LIN {X 2.525,Y 79.377,Z 54.000,A 180.000,B 0.000,C 180.000} C_DIS
LIN {X 2.581,Y 80.986,Z 54.000,A 180.000,B 0.000,C 180.000} C_DIS
LIN {X 2.591,Y 81.165,Z 54.000,A 180.000,B 0.000,C 180.000} C_DIS
LIN {X 2.675,Y 82.595,Z 54.000,A 180.000,B 0.000,C 180.000} C_DIS
LIN {X 2.685,Y 82.761,Z 54.000,A 180.000,B 0.000,C 180.000} C_DIS
LIN {X 2.686,Y 82.774,Z 54.000,A 180.000,B 0.000,C 180.000} C_DIS
LIN {X 2.700,Y 82.952,Z 54.000,A 180.000,B 0.000,C 180.000} C_DIS
LIN {X 2.818,Y 84.383,Z 54.000,A 180.000,B 0.000,C 180.000} C_DIS
LIN {X 2.833,Y 84.561,Z 54.000,A 180.000,B 0.000,C 180.000} C_DIS
LIN {X 3.004,Y 86.170,Z 54.000,A 180.000,B 0.000,C 180.000} C_DIS
LIN {X 3.025,Y 86.349,Z 54.000,A 180.000,B 0.000,C 180.000} C_DIS
LIN {X 3.233,Y 87.958,Z 54.000,A 180.000,B 0.000,C 180.000} C_DIS
LIN {X 3.259,Y 88.137,Z 54.000,A 180.000,B 0.000,C 180.000} C_DIS
LIN {X 3.479,Y 89.567,Z 54.000,A 180.000,B 0.000,C 180.000} C_DIS
LIN {X 3.506,Y 89.746,Z 54.000,A 180.000,B 0.000,C 180.000} C_DIS
LIN {X 3.538,Y 89.925,Z 54.000,A 180.000,B 0.000,C 180.000} C_DIS
LIN {X 3.792,Y 91.355,Z 54.000,A 180.000,B 0.000,C 180.000} C_DIS
LIN {X 3.825,Y 91.533,Z 54.000,A 180.000,B 0.000,C 180.000} C_DIS
LIN {X 4.150,Y 93.142,Z 54.000,A 180.000,B 0.000,C 180.000} C_DIS
LIN {X 4.189,Y 93.321,Z 54.000,A 180.000,B 0.000,C 180.000} C_DIS
LIN {X 4.513,Y 94.751,Z 54.000,A 180.000,B 0.000,C 180.000} C_DIS
LIN {X 4.554,Y 94.930,Z 54.000,A 180.000,B 0.000,C 180.000} C_DIS
LIN {X 4.598,Y 95.109,Z 54.000,A 180.000,B 0.000,C 180.000} C_DIS
LIN {X 4.958,Y 96.539,Z 54.000,A 180.000,B 0.000,C 180.000} C_DIS
LIN {X 5.005,Y 96.718,Z 54.000,A 180.000,B 0.000,C 180.000} C_DIS
LIN {X 5.400,Y 98.148,Z 54.000,A 180.000,B 0.000,C 180.000} C_DIS
LIN {X 5.450,Y 98.327,Z 54.000,A 180.000,B 0.000,C 180.000} C_DIS
LIN {X 5.503,Y 98.505,Z 54.000,A 180.000,B 0.000,C 180.000} C_DIS
LIN {X 5.935,Y 99.936,Z 54.000,A 180.000,B 0.000,C 180.000} C_DIS
LIN {X 5.992,Y 100.114,Z 54.000,A 180.000,B 0.000,C 180.000} C_DIS
LIN {X 6.460,Y 101.545,Z 54.000,A 180.000,B 0.000,C 180.000} C_DIS
LIN {X 6.520,Y 101.723,Z 54.000,A 180.000,B 0.000,C 180.000} C_DIS
LIN {X 7.026,Y 103.153,Z 54.000,A 180.000,B 0.000,C 180.000} C_DIS
LIN {X 7.089,Y 103.332,Z 54.000,A 180.000,B 0.000,C 180.000} C_DIS
LIN {X 7.154,Y 103.504,Z 54.000,A 180.000,B 0.000,C 180.000} C_DIS
LIN {X 7.701,Y 104.941,Z 54.000,A 180.000,B 0.000,C 180.000} C_DIS
LIN {X 7.773,Y 105.120,Z 54.000,A 180.000,B 0.000,C 180.000} C_DIS
LIN {X 8.355,Y 106.550,Z 54.000,A 180.000,B 0.000,C 180.000} C_DIS
LIN {X 8.405,Y 106.669,Z 54.000,A 180.000,B 0.000,C 180.000} C_DIS
LIN {X 9.053,Y 108.159,Z 54.000,A 180.000,B 0.000,C 180.000} C_DIS
LIN {X 9.120,Y 108.308,Z 54.000,A 180.000,B 0.000,C 180.000} C_DIS
LIN {X 9.797,Y 109.768,Z 54.000,A 180.000,B 0.000,C 180.000} C_DIS
LIN {X 9.836,Y 109.849,Z 54.000,A 180.000,B 0.000,C 180.000} C_DIS
LIN {X 10.551,Y 111.303,Z 54.000,A 180.000,B 0.000,C 180.000} C_DIS
LIN {X 10.587,Y 111.377,Z 54.000,A 180.000,B 0.000,C 180.000} C_DIS
LIN {X 10.680,Y 111.556,Z 54.000,A 180.000,B 0.000,C 180.000} C_DIS
LIN {X 11.332,Y 112.807,Z 54.000,A 180.000,B 0.000,C 180.000} C_DIS
LIN {X 11.426,Y 112.986,Z 54.000,A 180.000,B 0.000,C 180.000} C_DIS
LIN {X 12.215,Y 114.416,Z 54.000,A 180.000,B 0.000,C 180.000} C_DIS
LIN {X 12.317,Y 114.595,Z 54.000,A 180.000,B 0.000,C 180.000} C_DIS
LIN {X 13.053,Y 115.859,Z 54.000,A 180.000,B 0.000,C 180.000} C_DIS
LIN {X 13.151,Y 116.025,Z 54.000,A 180.000,B 0.000,C 180.000} C_DIS
LIN {X 13.232,Y 116.158,Z 54.000,A 180.000,B 0.000,C 180.000} C_DIS
LIN {X 14.029,Y 117.455,Z 54.000,A 180.000,B 0.000,C 180.000} C_DIS
LIN {X 14.126,Y 117.607,Z 54.000,A 180.000,B 0.000,C 180.000} C_DIS
LIN {X 14.953,Y 118.885,Z 54.000,A 180.000,B 0.000,C 180.000} C_DIS
LIN {X 15.020,Y 118.988,Z 54.000,A 180.000,B 0.000,C 180.000} C_DIS
LIN {X 15.072,Y 119.064,Z 54.000,A 180.000,B 0.000,C 180.000} C_DIS
LIN {X 15.924,Y 120.315,Z 54.000,A 180.000,B 0.000,C 180.000} C_DIS
LIN {X 16.047,Y 120.494,Z 54.000,A 180.000,B 0.000,C 180.000} C_DIS
LIN {X 16.986,Y 121.806,Z 54.000,A 180.000,B 0.000,C 180.000} C_DIS
LIN {X 17.073,Y 121.924,Z 54.000,A 180.000,B 0.000,C 180.000} C_DIS
LIN {X 18.059,Y 123.235,Z 54.000,A 180.000,B 0.000,C 180.000} C_DIS
LIN {X 18.152,Y 123.354,Z 54.000,A 180.000,B 0.000,C 180.000} C_DIS
LIN {X 19.139,Y 124.606,Z 54.000,A 180.000,B 0.000,C 180.000} C_DIS
LIN {X 19.286,Y 124.785,Z 54.000,A 180.000,B 0.000,C 180.000} C_DIS
LIN {X 20.204,Y 125.894,Z 54.000,A 180.000,B 0.000,C 180.000} C_DIS
LIN {X 20.323,Y 126.036,Z 54.000,A 180.000,B 0.000,C 180.000} C_DIS
LIN {X 21.410,Y 127.287,Z 54.000,A 180.000,B 0.000,C 180.000} C_DIS
LIN {X 21.456,Y 127.340,Z 54.000,A 180.000,B 0.000,C 180.000} C_DIS
LIN {X 21.570,Y 127.466,Z 54.000,A 180.000,B 0.000,C 180.000} C_DIS
LIN {X 22.547,Y 128.539,Z 54.000,A 180.000,B 0.000,C 180.000} C_DIS
LIN {X 22.707,Y 128.711,Z 54.000,A 180.000,B 0.000,C 180.000} C_DIS
LIN {X 23.780,Y 129.835,Z 54.000,A 180.000,B 0.000,C 180.000} C_DIS
LIN {X 23.910,Y 129.969,Z 54.000,A 180.000,B 0.000,C 180.000} C_DIS
LIN {X 25.031,Y 131.090,Z 54.000,A 180.000,B 0.000,C 180.000} C_DIS
LIN {X 25.165,Y 131.220,Z 54.000,A 180.000,B 0.000,C 180.000} C_DIS
LIN {X 26.289,Y 132.293,Z 54.000,A 180.000,B 0.000,C 180.000} C_DIS
LIN {X 26.461,Y 132.453,Z 54.000,A 180.000,B 0.000,C 180.000} C_DIS
LIN {X 27.534,Y 133.430,Z 54.000,A 180.000,B 0.000,C 180.000} C_DIS
LIN {X 27.660,Y 133.544,Z 54.000,A 180.000,B 0.000,C 180.000} C_DIS
LIN {X 27.713,Y 133.590,Z 54.000,A 180.000,B 0.000,C 180.000} C_DIS
LIN {X 28.964,Y 134.677,Z 54.000,A 180.000,B 0.000,C 180.000} C_DIS
LIN {X 29.106,Y 134.796,Z 54.000,A 180.000,B 0.000,C 180.000} C_DIS
LIN {X 30.215,Y 135.714,Z 54.000,A 180.000,B 0.000,C 180.000} C_DIS
LIN {X 30.394,Y 135.861,Z 54.000,A 180.000,B 0.000,C 180.000} C_DIS
LIN {X 31.646,Y 136.848,Z 54.000,A 180.000,B 0.000,C 180.000} C_DIS
LIN {X 31.765,Y 136.941,Z 54.000,A 180.000,B 0.000,C 180.000} C_DIS
LIN {X 33.076,Y 137.927,Z 54.000,A 180.000,B 0.000,C 180.000} C_DIS
LIN {X 33.194,Y 138.014,Z 54.000,A 180.000,B 0.000,C 180.000} C_DIS
LIN {X 34.506,Y 138.953,Z 54.000,A 180.000,B 0.000,C 180.000} C_DIS
LIN {X 34.685,Y 139.076,Z 54.000,A 180.000,B 0.000,C 180.000} C_DIS
LIN {X 35.936,Y 139.928,Z 54.000,A 180.000,B 0.000,C 180.000} C_DIS
LIN {X 36.012,Y 139.980,Z 54.000,A 180.000,B 0.000,C 180.000} C_DIS
LIN {X 36.115,Y 140.047,Z 54.000,A 180.000,B 0.000,C 180.000} C_DIS
LIN {X 37.393,Y 140.874,Z 54.000,A 180.000,B 0.000,C 180.000} C_DIS
LIN {X 37.545,Y 140.971,Z 54.000,A 180.000,B 0.000,C 180.000} C_DIS
LIN {X 38.842,Y 141.768,Z 54.000,A 180.000,B 0.000,C 180.000} C_DIS
LIN {X 38.975,Y 141.849,Z 54.000,A 180.000,B 0.000,C 180.000} C_DIS
LIN {X 39.141,Y 141.947,Z 54.000,A 180.000,B 0.000,C 180.000} C_DIS
LIN {X 40.405,Y 142.683,Z 54.000,A 180.000,B 0.000,C 180.000} C_DIS
LIN {X 40.584,Y 142.785,Z 54.000,A 180.000,B 0.000,C 180.000} C_DIS
LIN {X 42.014,Y 143.574,Z 54.000,A 180.000,B 0.000,C 180.000} C_DIS
LIN {X 42.193,Y 143.668,Z 54.000,A 180.000,B 0.000,C 180.000} C_DIS
LIN {X 43.444,Y 144.320,Z 54.000,A 180.000,B 0.000,C 180.000} C_DIS
LIN {X 43.623,Y 144.413,Z 54.000,A 180.000,B 0.000,C 180.000} C_DIS
LIN {X 43.697,Y 144.449,Z 54.000,A 180.000,B 0.000,C 180.000} C_DIS
LIN {X 45.151,Y 145.164,Z 54.000,A 180.000,B 0.000,C 180.000} C_DIS
LIN {X 45.232,Y 145.203,Z 54.000,A 180.000,B 0.000,C 180.000} C_DIS
LIN {X 46.692,Y 145.880,Z 54.000,A 180.000,B 0.000,C 180.000} C_DIS
LIN {X 46.841,Y 145.947,Z 54.000,A 180.000,B 0.000,C 180.000} C_DIS
LIN {X 48.331,Y 146.595,Z 54.000,A 180.000,B 0.000,C 180.000} C_DIS
LIN {X 48.450,Y 146.645,Z 54.000,A 180.000,B 0.000,C 180.000} C_DIS
LIN {X 49.880,Y 147.227,Z 54.000,A 180.000,B 0.000,C 180.000} C_DIS
LIN {X 50.059,Y 147.299,Z 54.000,A 180.000,B 0.000,C 180.000} C_DIS
LIN {X 51.496,Y 147.846,Z 54.000,A 180.000,B 0.000,C 180.000} C_DIS
LIN {X 51.668,Y 147.911,Z 54.000,A 180.000,B 0.000,C 180.000} C_DIS
LIN {X 51.847,Y 147.974,Z 54.000,A 180.000,B 0.000,C 180.000} C_DIS
LIN {X 53.277,Y 148.480,Z 54.000,A 180.000,B 0.000,C 180.000} C_DIS
LIN {X 53.455,Y 148.540,Z 54.000,A 180.000,B 0.000,C 180.000} C_DIS
LIN {X 54.290,Y 148.813,Z 54.000,A 180.000,B 0.000,C 180.000} C_DIS
LIN {X 54.886,Y 149.008,Z 54.000,A 180.000,B 0.000,C 180.000} C_DIS
LIN {X 55.064,Y 149.065,Z 54.000,A 180.000,B 0.000,C 180.000} C_DIS
LIN {X 56.495,Y 149.497,Z 54.000,A 180.000,B 0.000,C 180.000} C_DIS
LIN {X 56.673,Y 149.550,Z 54.000,A 180.000,B 0.000,C 180.000} C_DIS
LIN {X 56.852,Y 149.600,Z 54.000,A 180.000,B 0.000,C 180.000} C_DIS
LIN {X 58.282,Y 149.995,Z 54.000,A 180.000,B 0.000,C 180.000} C_DIS
LIN {X 58.461,Y 150.042,Z 54.000,A 180.000,B 0.000,C 180.000} C_DIS
LIN {X 59.891,Y 150.402,Z 54.000,A 180.000,B 0.000,C 180.000} C_DIS
LIN {X 60.070,Y 150.447,Z 54.000,A 180.000,B 0.000,C 180.000} C_DIS
LIN {X 60.249,Y 150.487,Z 54.000,A 180.000,B 0.000,C 180.000} C_DIS
LIN {X 61.679,Y 150.811,Z 54.000,A 180.000,B 0.000,C 180.000} C_DIS
LIN {X 61.858,Y 150.850,Z 54.000,A 180.000,B 0.000,C 180.000} C_DIS
LIN {X 63.467,Y 151.175,Z 54.000,A 180.000,B 0.000,C 180.000} C_DIS
LIN {X 63.645,Y 151.208,Z 54.000,A 180.000,B 0.000,C 180.000} C_DIS
LIN {X 65.075,Y 151.462,Z 54.000,A 180.000,B 0.000,C 180.000} C_DIS
LIN {X 65.254,Y 151.494,Z 54.000,A 180.000,B 0.000,C 180.000} C_DIS
LIN {X 65.433,Y 151.521,Z 54.000,A 180.000,B 0.000,C 180.000} C_DIS
LIN {X 66.863,Y 151.741,Z 54.000,A 180.000,B 0.000,C 180.000} C_DIS
LIN {X 67.042,Y 151.767,Z 54.000,A 180.000,B 0.000,C 180.000} C_DIS
LIN {X 68.651,Y 151.975,Z 54.000,A 180.000,B 0.000,C 180.000} C_DIS
LIN {X 68.830,Y 151.996,Z 54.000,A 180.000,B 0.000,C 180.000} C_DIS
LIN {X 70.439,Y 152.167,Z 54.000,A 180.000,B 0.000,C 180.000} C_DIS
LIN {X 70.617,Y 152.182,Z 54.000,A 180.000,B 0.000,C 180.000} C_DIS
LIN {X 72.048,Y 152.300,Z 54.000,A 180.000,B 0.000,C 180.000} C_DIS
LIN {X 72.226,Y 152.314,Z 54.000,A 180.000,B 0.000,C 180.000} C_DIS
LIN {X 72.239,Y 152.315,Z 54.000,A 180.000,B 0.000,C 180.000} C_DIS
LIN {X 72.405,Y 152.325,Z 54.000,A 180.000,B 0.000,C 180.000} C_DIS
LIN {X 73.835,Y 152.409,Z 54.000,A 180.000,B 0.000,C 180.000} C_DIS
LIN {X 74.014,Y 152.419,Z 54.000,A 180.000,B 0.000,C 180.000} C_DIS
LIN {X 75.623,Y 152.475,Z 54.000,A 180.000,B 0.000,C 180.000} C_DIS
LIN {X 75.802,Y 152.480,Z 54.000,A 180.000,B 0.000,C 180.000} C_DIS
LIN {X 77.411,Y 152.499,Z 54.000,A 180.000,B 0.000,C 180.000} C_DIS
LIN {X 77.589,Y 152.499,Z 54.000,A 180.000,B 0.000,C 180.000} C_DIS
LIN {X 79.198,Y 152.480,Z 54.000,A 180.000,B 0.000,C 180.000} C_DIS
LIN {X 79.377,Y 152.475,Z 54.000,A 180.000,B 0.000,C 180.000} C_DIS
LIN {X 80.986,Y 152.419,Z 54.000,A 180.000,B 0.000,C 180.000} C_DIS
LIN {X 81.165,Y 152.409,Z 54.000,A 180.000,B 0.000,C 180.000} C_DIS
LIN {X 82.595,Y 152.325,Z 54.000,A 180.000,B 0.000,C 180.000} C_DIS
LIN {X 82.761,Y 152.315,Z 54.000,A 180.000,B 0.000,C 180.000} C_DIS
LIN {X 82.774,Y 152.314,Z 54.000,A 180.000,B 0.000,C 180.000} C_DIS
LIN {X 82.952,Y 152.300,Z 54.000,A 180.000,B 0.000,C 180.000} C_DIS
LIN {X 84.383,Y 152.182,Z 54.000,A 180.000,B 0.000,C 180.000} C_DIS
LIN {X 84.561,Y 152.167,Z 54.000,A 180.000,B 0.000,C 180.000} C_DIS
LIN {X 86.170,Y 151.996,Z 54.000,A 180.000,B 0.000,C 180.000} C_DIS
LIN {X 86.349,Y 151.975,Z 54.000,A 180.000,B 0.000,C 180.000} C_DIS
LIN {X 87.958,Y 151.767,Z 54.000,A 180.000,B 0.000,C 180.000} C_DIS
LIN {X 88.137,Y 151.741,Z 54.000,A 180.000,B 0.000,C 180.000} C_DIS
LIN {X 89.567,Y 151.521,Z 54.000,A 180.000,B 0.000,C 180.000} C_DIS
LIN {X 89.746,Y 151.494,Z 54.000,A 180.000,B 0.000,C 180.000} C_DIS
LIN {X 89.925,Y 151.462,Z 54.000,A 180.000,B 0.000,C 180.000} C_DIS
LIN {X 91.355,Y 151.208,Z 54.000,A 180.000,B 0.000,C 180.000} C_DIS
LIN {X 91.533,Y 151.175,Z 54.000,A 180.000,B 0.000,C 180.000} C_DIS
LIN {X 93.142,Y 150.850,Z 54.000,A 180.000,B 0.000,C 180.000} C_DIS
LIN {X 93.321,Y 150.811,Z 54.000,A 180.000,B 0.000,C 180.000} C_DIS
LIN {X 94.751,Y 150.487,Z 54.000,A 180.000,B 0.000,C 180.000} C_DIS
LIN {X 94.930,Y 150.447,Z 54.000,A 180.000,B 0.000,C 180.000} C_DIS
LIN {X 95.109,Y 150.402,Z 54.000,A 180.000,B 0.000,C 180.000} C_DIS
LIN {X 96.539,Y 150.042,Z 54.000,A 180.000,B 0.000,C 180.000} C_DIS
LIN {X 96.718,Y 149.995,Z 54.000,A 180.000,B 0.000,C 180.000} C_DIS
LIN {X 98.148,Y 149.600,Z 54.000,A 180.000,B 0.000,C 180.000} C_DIS
LIN {X 98.327,Y 149.550,Z 54.000,A 180.000,B 0.000,C 180.000} C_DIS
LIN {X 98.505,Y 149.497,Z 54.000,A 180.000,B 0.000,C 180.000} C_DIS
LIN {X 99.936,Y 149.065,Z 54.000,A 180.000,B 0.000,C 180.000} C_DIS
LIN {X 100.114,Y 149.008,Z 54.000,A 180.000,B 0.000,C 180.000} C_DIS
LIN {X 101.545,Y 148.540,Z 54.000,A 180.000,B 0.000,C 180.000} C_DIS
LIN {X 101.723,Y 148.480,Z 54.000,A 180.000,B 0.000,C 180.000} C_DIS
LIN {X 103.153,Y 147.974,Z 54.000,A 180.000,B 0.000,C 180.000} C_DIS
LIN {X 103.332,Y 147.911,Z 54.000,A 180.000,B 0.000,C 180.000} C_DIS
LIN {X 103.504,Y 147.846,Z 54.000,A 180.000,B 0.000,C 180.000} C_DIS
LIN {X 104.941,Y 147.299,Z 54.000,A 180.000,B 0.000,C 180.000} C_DIS
LIN {X 105.120,Y 147.227,Z 54.000,A 180.000,B 0.000,C 180.000} C_DIS
LIN {X 106.550,Y 146.645,Z 54.000,A 180.000,B 0.000,C 180.000} C_DIS
LIN {X 106.669,Y 146.595,Z 54.000,A 180.000,B 0.000,C 180.000} C_DIS
LIN {X 108.159,Y 145.947,Z 54.000,A 180.000,B 0.000,C 180.000} C_DIS
LIN {X 108.308,Y 145.880,Z 54.000,A 180.000,B 0.000,C 180.000} C_DIS
LIN {X 109.768,Y 145.203,Z 54.000,A 180.000,B 0.000,C 180.000} C_DIS
LIN {X 109.849,Y 145.164,Z 54.000,A 180.000,B 0.000,C 180.000} C_DIS
LIN {X 111.303,Y 144.449,Z 54.000,A 180.000,B 0.000,C 180.000} C_DIS
LIN {X 111.377,Y 144.413,Z 54.000,A 180.000,B 0.000,C 180.000} C_DIS
LIN {X 111.556,Y 144.320,Z 54.000,A 180.000,B 0.000,C 180.000} C_DIS
LIN {X 112.807,Y 143.668,Z 54.000,A 180.000,B 0.000,C 180.000} C_DIS
LIN {X 112.986,Y 143.574,Z 54.000,A 180.000,B 0.000,C 180.000} C_DIS
LIN {X 114.416,Y 142.785,Z 54.000,A 180.000,B 0.000,C 180.000} C_DIS
LIN {X 114.595,Y 142.683,Z 54.000,A 180.000,B 0.000,C 180.000} C_DIS
LIN {X 115.859,Y 141.947,Z 54.000,A 180.000,B 0.000,C 180.000} C_DIS
LIN {X 116.025,Y 141.849,Z 54.000,A 180.000,B 0.000,C 180.000} C_DIS
LIN {X 116.158,Y 141.768,Z 54.000,A 180.000,B 0.000,C 180.000} C_DIS
LIN {X 117.455,Y 140.971,Z 54.000,A 180.000,B 0.000,C 180.000} C_DIS
LIN {X 117.607,Y 140.874,Z 54.000,A 180.000,B 0.000,C 180.000} C_DIS
LIN {X 118.885,Y 140.047,Z 54.000,A 180.000,B 0.000,C 180.000} C_DIS
LIN {X 118.988,Y 139.980,Z 54.000,A 180.000,B 0.000,C 180.000} C_DIS
LIN {X 119.064,Y 139.928,Z 54.000,A 180.000,B 0.000,C 180.000} C_DIS
LIN {X 120.315,Y 139.076,Z 54.000,A 180.000,B 0.000,C 180.000} C_DIS
LIN {X 120.494,Y 138.953,Z 54.000,A 180.000,B 0.000,C 180.000} C_DIS
LIN {X 121.806,Y 138.014,Z 54.000,A 180.000,B 0.000,C 180.000} C_DIS
LIN {X 121.924,Y 137.927,Z 54.000,A 180.000,B 0.000,C 180.000} C_DIS
LIN {X 122.641,Y 137.388,Z 54.000,A 180.000,B 0.000,C 180.000} C_DIS
; Link Move Starts
LIN {X 122.893,Y 137.199,Z 54.000,A 180.000,B 0.000,C 180.000} C_DIS
LIN {X 123.144,Y 137.009,Z 53.999,A 180.000,B 0.000,C 180.000} C_DIS
LIN {X 123.394,Y 136.817,Z 53.998,A 180.000,B 0.000,C 180.000} C_DIS
LIN {X 123.641,Y 136.622,Z 53.996,A 180.000,B 0.000,C 180.000} C_DIS
LIN {X 123.889,Y 136.427,Z 53.994,A 180.000,B 0.000,C 180.000} C_DIS
LIN {X 124.136,Y 136.232,Z 53.991,A 180.000,B 0.000,C 180.000} C_DIS
LIN {X 124.383,Y 136.036,Z 53.988,A 180.000,B 0.000,C 180.000} C_DIS
LIN {X 124.630,Y 135.841,Z 53.985,A 180.000,B 0.000,C 180.000} C_DIS
LIN {X 124.873,Y 135.641,Z 53.981,A 180.000,B 0.000,C 180.000} C_DIS
LIN {X 125.116,Y 135.440,Z 53.977,A 180.000,B 0.000,C 180.000} C_DIS
LIN {X 125.359,Y 135.239,Z 53.972,A 180.000,B 0.000,C 180.000} C_DIS
LIN {X 125.480,Y 135.139,Z 53.969,A 180.000,B 0.000,C 180.000} C_DIS
LIN {X 125.601,Y 135.038,Z 53.967,A 180.000,B 0.000,C 180.000} C_DIS
LIN {X 125.723,Y 134.938,Z 53.964,A 180.000,B 0.000,C 180.000} C_DIS
LIN {X 125.844,Y 134.837,Z 53.961,A 180.000,B 0.000,C 180.000} C_DIS
LIN {X 125.965,Y 134.737,Z 53.959,A 180.000,B 0.000,C 180.000} C_DIS
LIN {X 126.085,Y 134.635,Z 53.956,A 180.000,B 0.000,C 180.000} C_DIS
LIN {X 126.204,Y 134.531,Z 53.952,A 180.000,B 0.000,C 180.000} C_DIS
LIN {X 126.323,Y 134.428,Z 53.949,A 180.000,B 0.000,C 180.000} C_DIS
LIN {X 126.442,Y 134.325,Z 53.946,A 180.000,B 0.000,C 180.000} C_DIS
LIN {X 126.561,Y 134.222,Z 53.943,A 180.000,B 0.000,C 180.000} C_DIS
LIN {X 126.680,Y 134.118,Z 53.939,A 180.000,B 0.000,C 180.000} C_DIS
LIN {X 126.798,Y 134.015,Z 53.936,A 180.000,B 0.000,C 180.000} C_DIS
LIN {X 126.917,Y 133.912,Z 53.932,A 180.000,B 0.000,C 180.000} C_DIS
LIN {X 127.036,Y 133.808,Z 53.928,A 180.000,B 0.000,C 180.000} C_DIS
LIN {X 127.155,Y 133.705,Z 53.925,A 180.000,B 0.000,C 180.000} C_DIS
LIN {X 127.274,Y 133.602,Z 53.921,A 180.000,B 0.000,C 180.000} C_DIS
LIN {X 127.392,Y 133.497,Z 53.917,A 180.000,B 0.000,C 180.000} C_DIS
LIN {X 127.508,Y 133.391,Z 53.913,A 180.000,B 0.000,C 180.000} C_DIS
LIN {X 127.625,Y 133.285,Z 53.909,A 180.000,B 0.000,C 180.000} C_DIS
LIN {X 127.741,Y 133.179,Z 53.905,A 180.000,B 0.000,C 180.000} C_DIS
LIN {X 127.858,Y 133.073,Z 53.900,A 180.000,B 0.000,C 180.000} C_DIS
LIN {X 127.974,Y 132.967,Z 53.896,A 180.000,B 0.000,C 180.000} C_DIS
LIN {X 128.091,Y 132.861,Z 53.892,A 180.000,B 0.000,C 180.000} C_DIS
LIN {X 128.207,Y 132.755,Z 53.887,A 180.000,B 0.000,C 180.000} C_DIS
LIN {X 128.324,Y 132.649,Z 53.883,A 180.000,B 0.000,C 180.000} C_DIS
LIN {X 128.440,Y 132.543,Z 53.878,A 180.000,B 0.000,C 180.000} C_DIS
LIN {X 128.557,Y 132.437,Z 53.873,A 180.000,B 0.000,C 180.000} C_DIS
LIN {X 128.672,Y 132.330,Z 53.869,A 180.000,B 0.000,C 180.000} C_DIS
LIN {X 128.786,Y 132.221,Z 53.864,A 180.000,B 0.000,C 180.000} C_DIS
LIN {X 128.900,Y 132.113,Z 53.859,A 180.000,B 0.000,C 180.000} C_DIS
LIN {X 129.014,Y 132.004,Z 53.854,A 180.000,B 0.000,C 180.000} C_DIS
LIN {X 129.071,Y 131.950,Z 53.851,A 180.000,B 0.000,C 180.000} C_DIS
LIN {X 129.128,Y 131.895,Z 53.849,A 180.000,B 0.000,C 180.000} C_DIS
LIN {X 129.185,Y 131.841,Z 53.846,A 180.000,B 0.000,C 180.000} C_DIS
LIN {X 129.242,Y 131.787,Z 53.844,A 180.000,B 0.000,C 180.000} C_DIS
LIN {X 129.299,Y 131.732,Z 53.841,A 180.000,B 0.000,C 180.000} C_DIS
LIN {X 129.356,Y 131.678,Z 53.839,A 180.000,B 0.000,C 180.000} C_DIS
LIN {X 129.413,Y 131.623,Z 53.836,A 180.000,B 0.000,C 180.000} C_DIS
LIN {X 129.527,Y 131.515,Z 53.831,A 180.000,B 0.000,C 180.000} C_DIS
LIN {X 129.641,Y 131.406,Z 53.825,A 180.000,B 0.000,C 180.000} C_DIS
LIN {X 129.755,Y 131.297,Z 53.820,A 180.000,B 0.000,C 180.000} C_DIS
LIN {X 129.869,Y 131.189,Z 53.815,A 180.000,B 0.000,C 180.000} C_DIS
LIN {X 129.925,Y 131.134,Z 53.812,A 180.000,B 0.000,C 180.000} C_DIS
LIN {X 130.092,Y 130.967,Z 53.804,A 180.000,B 0.000,C 180.000} C_DIS
LIN {X 130.204,Y 130.855,Z 53.798,A 180.000,B 0.000,C 180.000} C_DIS
LIN {X 130.259,Y 130.800,Z 53.796,A 180.000,B 0.000,C 180.000} C_DIS
LIN {X 130.371,Y 130.688,Z 53.790,A 180.000,B 0.000,C 180.000} C_DIS
LIN {X 130.538,Y 130.521,Z 53.782,A 180.000,B 0.000,C 180.000} C_DIS
LIN {X 130.649,Y 130.410,Z 53.776,A 180.000,B 0.000,C 180.000} C_DIS
LIN {X 130.705,Y 130.354,Z 53.774,A 180.000,B 0.000,C 180.000} C_DIS
LIN {X 130.816,Y 130.243,Z 53.768,A 180.000,B 0.000,C 180.000} C_DIS
LIN {X 130.983,Y 130.076,Z 53.760,A 180.000,B 0.000,C 180.000} C_DIS
LIN {X 131.095,Y 129.964,Z 53.754,A 180.000,B 0.000,C 180.000} C_DIS
LIN {X 131.150,Y 129.909,Z 53.752,A 180.000,B 0.000,C 180.000} C_DIS
LIN {X 131.205,Y 129.852,Z 53.749,A 180.000,B 0.000,C 180.000} C_DIS
LIN {X 131.313,Y 129.738,Z 53.743,A 180.000,B 0.000,C 180.000} C_DIS
LIN {X 131.368,Y 129.681,Z 53.741,A 180.000,B 0.000,C 180.000} C_DIS
LIN {X 131.477,Y 129.567,Z 53.735,A 180.000,B 0.000,C 180.000} C_DIS
LIN {X 131.640,Y 129.396,Z 53.727,A 180.000,B 0.000,C 180.000} C_DIS
LIN {X 131.748,Y 129.282,Z 53.721,A 180.000,B 0.000,C 180.000} C_DIS
LIN {X 131.803,Y 129.225,Z 53.719,A 180.000,B 0.000,C 180.000} C_DIS
LIN {X 131.911,Y 129.111,Z 53.713,A 180.000,B 0.000,C 180.000} C_DIS
LIN {X 132.238,Y 128.769,Z 53.697,A 180.000,B 0.000,C 180.000} C_DIS
LIN {X 132.346,Y 128.655,Z 53.691,A 180.000,B 0.000,C 180.000} C_DIS
LIN {X 132.400,Y 128.597,Z 53.688,A 180.000,B 0.000,C 180.000} C_DIS
LIN {X 132.453,Y 128.539,Z 53.686,A 180.000,B 0.000,C 180.000} C_DIS
LIN {X 132.559,Y 128.423,Z 53.680,A 180.000,B 0.000,C 180.000} C_DIS
LIN {X 132.877,Y 128.073,Z 53.664,A 180.000,B 0.000,C 180.000} C_DIS
LIN {X 133.036,Y 127.899,Z 53.655,A 180.000,B 0.000,C 180.000} C_DIS
LIN {X 133.142,Y 127.782,Z 53.650,A 180.000,B 0.000,C 180.000} C_DIS
LIN {X 133.460,Y 127.433,Z 53.633,A 180.000,B 0.000,C 180.000} C_DIS
LIN {X 133.513,Y 127.375,Z 53.631,A 180.000,B 0.000,C 180.000} C_DIS
LIN {X 133.566,Y 127.316,Z 53.628,A 180.000,B 0.000,C 180.000} C_DIS
LIN {X 133.824,Y 127.019,Z 53.614,A 180.000,B 0.000,C 180.000} C_DIS
LIN {X 134.340,Y 126.424,Z 53.587,A 180.000,B 0.000,C 180.000} C_DIS
LIN {X 134.598,Y 126.127,Z 53.573,A 180.000,B 0.000,C 180.000} C_DIS
LIN {X 134.650,Y 126.067,Z 53.570,A 180.000,B 0.000,C 180.000} C_DIS
LIN {X 134.701,Y 126.008,Z 53.567,A 180.000,B 0.000,C 180.000} C_DIS
LIN {X 134.752,Y 125.947,Z 53.565,A 180.000,B 0.000,C 180.000} C_DIS
LIN {X 135.053,Y 125.583,Z 53.548,A 180.000,B 0.000,C 180.000} C_DIS
LIN {X 135.807,Y 124.673,Z 53.507,A 180.000,B 0.000,C 180.000} C_DIS
LIN {X 135.856,Y 124.612,Z 53.504,A 180.000,B 0.000,C 180.000} C_DIS
LIN {X 136.880,Y 123.314,Z 53.446,A 180.000,B 0.000,C 180.000} C_DIS
LIN {X 136.929,Y 123.252,Z 53.444,A 180.000,B 0.000,C 180.000} C_DIS
LIN {X 137.213,Y 122.874,Z 53.427,A 180.000,B 0.000,C 180.000} C_DIS
LIN {X 137.923,Y 121.930,Z 53.386,A 180.000,B 0.000,C 180.000} C_DIS
LIN {X 137.970,Y 121.867,Z 53.383,A 180.000,B 0.000,C 180.000} C_DIS
LIN {X 138.016,Y 121.803,Z 53.380,A 180.000,B 0.000,C 180.000} C_DIS
LIN {X 138.107,Y 121.675,Z 53.375,A 180.000,B 0.000,C 180.000} C_DIS
LIN {X 138.382,Y 121.291,Z 53.358,A 180.000,B 0.000,C 180.000} C_DIS
LIN {X 138.474,Y 121.162,Z 53.353,A 180.000,B 0.000,C 180.000} C_DIS
LIN {X 138.749,Y 120.778,Z 53.336,A 180.000,B 0.000,C 180.000} C_DIS
LIN {X 138.795,Y 120.714,Z 53.334,A 180.000,B 0.000,C 180.000} C_DIS
LIN {X 138.887,Y 120.586,Z 53.328,A 180.000,B 0.000,C 180.000} C_DIS
LIN {X 138.978,Y 120.458,Z 53.323,A 180.000,B 0.000,C 180.000} C_DIS
LIN {X 139.023,Y 120.393,Z 53.320,A 180.000,B 0.000,C 180.000} C_DIS
LIN {X 139.112,Y 120.263,Z 53.314,A 180.000,B 0.000,C 180.000} C_DIS
LIN {X 139.156,Y 120.198,Z 53.312,A 180.000,B 0.000,C 180.000} C_DIS
LIN {X 139.245,Y 120.068,Z 53.306,A 180.000,B 0.000,C 180.000} C_DIS
LIN {X 139.511,Y 119.677,Z 53.290,A 180.000,B 0.000,C 180.000} C_DIS
LIN {X 139.599,Y 119.547,Z 53.284,A 180.000,B 0.000,C 180.000} C_DIS
LIN {X 139.732,Y 119.352,Z 53.276,A 180.000,B 0.000,C 180.000} C_DIS
LIN {X 139.821,Y 119.222,Z 53.270,A 180.000,B 0.000,C 180.000} C_DIS
LIN {X 139.865,Y 119.157,Z 53.268,A 180.000,B 0.000,C 180.000} C_DIS
LIN {X 139.954,Y 119.026,Z 53.262,A 180.000,B 0.000,C 180.000} C_DIS
LIN {X 139.998,Y 118.961,Z 53.259,A 180.000,B 0.000,C 180.000} C_DIS
LIN {X 140.040,Y 118.895,Z 53.257,A 180.000,B 0.000,C 180.000} C_DIS
LIN {X 140.126,Y 118.763,Z 53.251,A 180.000,B 0.000,C 180.000} C_DIS
LIN {X 140.254,Y 118.564,Z 53.243,A 180.000,B 0.000,C 180.000} C_DIS
LIN {X 140.340,Y 118.432,Z 53.237,A 180.000,B 0.000,C 180.000} C_DIS
LIN {X 140.383,Y 118.366,Z 53.235,A 180.000,B 0.000,C 180.000} C_DIS
LIN {X 140.468,Y 118.234,Z 53.229,A 180.000,B 0.000,C 180.000} C_DIS
LIN {X 140.597,Y 118.035,Z 53.221,A 180.000,B 0.000,C 180.000} C_DIS
LIN {X 140.682,Y 117.903,Z 53.215,A 180.000,B 0.000,C 180.000} C_DIS
LIN {X 140.725,Y 117.837,Z 53.213,A 180.000,B 0.000,C 180.000} C_DIS
LIN {X 140.811,Y 117.705,Z 53.207,A 180.000,B 0.000,C 180.000} C_DIS
LIN {X 140.896,Y 117.573,Z 53.202,A 180.000,B 0.000,C 180.000} C_DIS
LIN {X 140.939,Y 117.506,Z 53.199,A 180.000,B 0.000,C 180.000} C_DIS
LIN {X 140.980,Y 117.439,Z 53.196,A 180.000,B 0.000,C 180.000} C_DIS
LIN {X 141.063,Y 117.305,Z 53.191,A 180.000,B 0.000,C 180.000} C_DIS
LIN {X 141.145,Y 117.171,Z 53.185,A 180.000,B 0.000,C 180.000} C_DIS
LIN {X 141.228,Y 117.037,Z 53.180,A 180.000,B 0.000,C 180.000} C_DIS
LIN {X 141.310,Y 116.903,Z 53.174,A 180.000,B 0.000,C 180.000} C_DIS
LIN {X 141.392,Y 116.768,Z 53.169,A 180.000,B 0.000,C 180.000} C_DIS
LIN {X 141.475,Y 116.634,Z 53.164,A 180.000,B 0.000,C 180.000} C_DIS
LIN {X 141.516,Y 116.567,Z 53.161,A 180.000,B 0.000,C 180.000} C_DIS
LIN {X 141.557,Y 116.500,Z 53.159,A 180.000,B 0.000,C 180.000} C_DIS
LIN {X 141.599,Y 116.433,Z 53.156,A 180.000,B 0.000,C 180.000} C_DIS
LIN {X 141.640,Y 116.366,Z 53.154,A 180.000,B 0.000,C 180.000} C_DIS
LIN {X 141.681,Y 116.299,Z 53.151,A 180.000,B 0.000,C 180.000} C_DIS
LIN {X 141.722,Y 116.232,Z 53.148,A 180.000,B 0.000,C 180.000} C_DIS
LIN {X 141.805,Y 116.097,Z 53.143,A 180.000,B 0.000,C 180.000} C_DIS
LIN {X 141.886,Y 115.963,Z 53.139,A 180.000,B 0.000,C 180.000} C_DIS
LIN {X 141.965,Y 115.826,Z 53.134,A 180.000,B 0.000,C 180.000} C_DIS
LIN {X 142.045,Y 115.690,Z 53.129,A 180.000,B 0.000,C 180.000} C_DIS
LIN {X 142.124,Y 115.554,Z 53.124,A 180.000,B 0.000,C 180.000} C_DIS
LIN {X 142.203,Y 115.418,Z 53.120,A 180.000,B 0.000,C 180.000} C_DIS
LIN {X 142.282,Y 115.282,Z 53.115,A 180.000,B 0.000,C 180.000} C_DIS
LIN {X 142.362,Y 115.146,Z 53.110,A 180.000,B 0.000,C 180.000} C_DIS
LIN {X 142.441,Y 115.010,Z 53.106,A 180.000,B 0.000,C 180.000} C_DIS
LIN {X 142.520,Y 114.874,Z 53.102,A 180.000,B 0.000,C 180.000} C_DIS
LIN {X 142.600,Y 114.738,Z 53.097,A 180.000,B 0.000,C 180.000} C_DIS
LIN {X 142.679,Y 114.602,Z 53.093,A 180.000,B 0.000,C 180.000} C_DIS
LIN {X 142.758,Y 114.465,Z 53.089,A 180.000,B 0.000,C 180.000} C_DIS
LIN {X 142.834,Y 114.327,Z 53.085,A 180.000,B 0.000,C 180.000} C_DIS
LIN {X 142.910,Y 114.189,Z 53.081,A 180.000,B 0.000,C 180.000} C_DIS
LIN {X 142.986,Y 114.051,Z 53.077,A 180.000,B 0.000,C 180.000} C_DIS
LIN {X 143.062,Y 113.914,Z 53.073,A 180.000,B 0.000,C 180.000} C_DIS
LIN {X 143.138,Y 113.776,Z 53.070,A 180.000,B 0.000,C 180.000} C_DIS
LIN {X 143.214,Y 113.638,Z 53.066,A 180.000,B 0.000,C 180.000} C_DIS
LIN {X 143.290,Y 113.500,Z 53.062,A 180.000,B 0.000,C 180.000} C_DIS
LIN {X 143.366,Y 113.362,Z 53.059,A 180.000,B 0.000,C 180.000} C_DIS
LIN {X 143.442,Y 113.224,Z 53.056,A 180.000,B 0.000,C 180.000} C_DIS
LIN {X 143.518,Y 113.086,Z 53.052,A 180.000,B 0.000,C 180.000} C_DIS
LIN {X 143.594,Y 112.948,Z 53.049,A 180.000,B 0.000,C 180.000} C_DIS
LIN {X 143.667,Y 112.808,Z 53.046,A 180.000,B 0.000,C 180.000} C_DIS
LIN {X 143.740,Y 112.669,Z 53.043,A 180.000,B 0.000,C 180.000} C_DIS
LIN {X 143.813,Y 112.529,Z 53.040,A 180.000,B 0.000,C 180.000} C_DIS
LIN {X 143.885,Y 112.390,Z 53.037,A 180.000,B 0.000,C 180.000} C_DIS
LIN {X 143.958,Y 112.250,Z 53.034,A 180.000,B 0.000,C 180.000} C_DIS
LIN {X 144.031,Y 112.110,Z 53.032,A 180.000,B 0.000,C 180.000} C_DIS
LIN {X 144.104,Y 111.971,Z 53.029,A 180.000,B 0.000,C 180.000} C_DIS
LIN {X 144.177,Y 111.831,Z 53.027,A 180.000,B 0.000,C 180.000} C_DIS
LIN {X 144.322,Y 111.552,Z 53.022,A 180.000,B 0.000,C 180.000} C_DIS
LIN {X 144.465,Y 111.271,Z 53.018,A 180.000,B 0.000,C 180.000} C_DIS
LIN {X 144.604,Y 110.988,Z 53.014,A 180.000,B 0.000,C 180.000} C_DIS
LIN {X 144.743,Y 110.706,Z 53.011,A 180.000,B 0.000,C 180.000} C_DIS
LIN {X 144.882,Y 110.423,Z 53.008,A 180.000,B 0.000,C 180.000} C_DIS
LIN {X 145.021,Y 110.140,Z 53.005,A 180.000,B 0.000,C 180.000} C_DIS
LIN {X 145.160,Y 109.858,Z 53.003,A 180.000,B 0.000,C 180.000} C_DIS
LIN {X 145.294,Y 109.572,Z 53.002,A 180.000,B 0.000,C 180.000} C_DIS
LIN {X 145.426,Y 109.286,Z 53.001,A 180.000,B 0.000,C 180.000} C_DIS
LIN {X 145.559,Y 109.001,Z 53.000,A 180.000,B 0.000,C 180.000} C_DIS
LIN {X 145.656,Y 108.791,Z 53.000,A 180.000,B 0.000,C 180.000} C_DIS
; Cutting Move Starts
LIN {X 145.880,Y 108.308,Z 53.000,A 180.000,B 0.000,C 180.000} C_DIS
LIN {X 145.947,Y 108.159,Z 53.000,A 180.000,B 0.000,C 180.000} C_DIS
LIN {X 146.595,Y 106.669,Z 53.000,A 180.000,B 0.000,C 180.000} C_DIS
LIN {X 146.645,Y 106.550,Z 53.000,A 180.000,B 0.000,C 180.000} C_DIS
LIN {X 147.227,Y 105.120,Z 53.000,A 180.000,B 0.000,C 180.000} C_DIS
LIN {X 147.299,Y 104.941,Z 53.000,A 180.000,B 0.000,C 180.000} C_DIS
LIN {X 147.846,Y 103.504,Z 53.000,A 180.000,B 0.000,C 180.000} C_DIS
LIN {X 147.911,Y 103.332,Z 53.000,A 180.000,B 0.000,C 180.000} C_DIS
LIN {X 147.974,Y 103.153,Z 53.000,A 180.000,B 0.000,C 180.000} C_DIS
LIN {X 148.480,Y 101.723,Z 53.000,A 180.000,B 0.000,C 180.000} C_DIS
LIN {X 148.540,Y 101.545,Z 53.000,A 180.000,B 0.000,C 180.000} C_DIS
LIN {X 149.008,Y 100.114,Z 53.000,A 180.000,B 0.000,C 180.000} C_DIS
LIN {X 149.065,Y 99.936,Z 53.000,A 180.000,B 0.000,C 180.000} C_DIS
LIN {X 149.497,Y 98.505,Z 53.000,A 180.000,B 0.000,C 180.000} C_DIS
LIN {X 149.550,Y 98.327,Z 53.000,A 180.000,B 0.000,C 180.000} C_DIS
LIN {X 149.600,Y 98.148,Z 53.000,A 180.000,B 0.000,C 180.000} C_DIS
LIN {X 149.995,Y 96.718,Z 53.000,A 180.000,B 0.000,C 180.000} C_DIS
LIN {X 150.042,Y 96.539,Z 53.000,A 180.000,B 0.000,C 180.000} C_DIS
LIN {X 150.402,Y 95.109,Z 53.000,A 180.000,B 0.000,C 180.000} C_DIS
LIN {X 150.447,Y 94.930,Z 53.000,A 180.000,B 0.000,C 180.000} C_DIS
LIN {X 150.487,Y 94.751,Z 53.000,A 180.000,B 0.000,C 180.000} C_DIS
LIN {X 150.811,Y 93.321,Z 53.000,A 180.000,B 0.000,C 180.000} C_DIS
LIN {X 150.850,Y 93.142,Z 53.000,A 180.000,B 0.000,C 180.000} C_DIS
LIN {X 151.175,Y 91.533,Z 53.000,A 180.000,B 0.000,C 180.000} C_DIS
LIN {X 151.208,Y 91.355,Z 53.000,A 180.000,B 0.000,C 180.000} C_DIS
LIN {X 151.462,Y 89.925,Z 53.000,A 180.000,B 0.000,C 180.000} C_DIS
LIN {X 151.494,Y 89.746,Z 53.000,A 180.000,B 0.000,C 180.000} C_DIS
LIN {X 151.521,Y 89.567,Z 53.000,A 180.000,B 0.000,C 180.000} C_DIS
LIN {X 151.741,Y 88.137,Z 53.000,A 180.000,B 0.000,C 180.000} C_DIS
LIN {X 151.767,Y 87.958,Z 53.000,A 180.000,B 0.000,C 180.000} C_DIS
LIN {X 151.975,Y 86.349,Z 53.000,A 180.000,B 0.000,C 180.000} C_DIS
LIN {X 151.996,Y 86.170,Z 53.000,A 180.000,B 0.000,C 180.000} C_DIS
LIN {X 152.167,Y 84.561,Z 53.000,A 180.000,B 0.000,C 180.000} C_DIS
LIN {X 152.182,Y 84.383,Z 53.000,A 180.000,B 0.000,C 180.000} C_DIS
LIN {X 152.300,Y 82.952,Z 53.000,A 180.000,B 0.000,C 180.000} C_DIS
LIN {X 152.314,Y 82.774,Z 53.000,A 180.000,B 0.000,C 180.000} C_DIS
LIN {X 152.315,Y 82.761,Z 53.000,A 180.000,B 0.000,C 180.000} C_DIS
LIN {X 152.325,Y 82.595,Z 53.000,A 180.000,B 0.000,C 180.000} C_DIS
LIN {X 152.409,Y 81.165,Z 53.000,A 180.000,B 0.000,C 180.000} C_DIS
LIN {X 152.419,Y 80.986,Z 53.000,A 180.000,B 0.000,C 180.000} C_DIS
LIN {X 152.475,Y 79.377,Z 53.000,A 180.000,B 0.000,C 180.000} C_DIS
LIN {X 152.480,Y 79.198,Z 53.000,A 180.000,B 0.000,C 180.000} C_DIS
LIN {X 152.499,Y 77.589,Z 53.000,A 180.000,B 0.000,C 180.000} C_DIS
LIN {X 152.499,Y 77.411,Z 53.000,A 180.000,B 0.000,C 180.000} C_DIS
LIN {X 152.480,Y 75.802,Z 53.000,A 180.000,B 0.000,C 180.000} C_DIS
LIN {X 152.475,Y 75.623,Z 53.000,A 180.000,B 0.000,C 180.000} C_DIS
LIN {X 152.419,Y 74.014,Z 53.000,A 180.000,B 0.000,C 180.000} C_DIS
LIN {X 152.409,Y 73.835,Z 53.000,A 180.000,B 0.000,C 180.000} C_DIS
LIN {X 152.325,Y 72.405,Z 53.000,A 180.000,B 0.000,C 180.000} C_DIS
LIN {X 152.315,Y 72.239,Z 53.000,A 180.000,B 0.000,C 180.000} C_DIS
LIN {X 152.314,Y 72.226,Z 53.000,A 180.000,B 0.000,C 180.000} C_DIS
LIN {X 152.300,Y 72.048,Z 53.000,A 180.000,B 0.000,C 180.000} C_DIS
LIN {X 152.182,Y 70.617,Z 53.000,A 180.000,B 0.000,C 180.000} C_DIS
LIN {X 152.167,Y 70.439,Z 53.000,A 180.000,B 0.000,C 180.000} C_DIS
LIN {X 151.996,Y 68.830,Z 53.000,A 180.000,B 0.000,C 180.000} C_DIS
LIN {X 151.975,Y 68.651,Z 53.000,A 180.000,B 0.000,C 180.000} C_DIS
LIN {X 151.767,Y 67.042,Z 53.000,A 180.000,B 0.000,C 180.000} C_DIS
LIN {X 151.741,Y 66.863,Z 53.000,A 180.000,B 0.000,C 180.000} C_DIS
LIN {X 151.521,Y 65.433,Z 53.000,A 180.000,B 0.000,C 180.000} C_DIS
LIN {X 151.494,Y 65.254,Z 53.000,A 180.000,B 0.000,C 180.000} C_DIS
LIN {X 151.462,Y 65.075,Z 53.000,A 180.000,B 0.000,C 180.000} C_DIS
LIN {X 151.208,Y 63.645,Z 53.000,A 180.000,B 0.000,C 180.000} C_DIS
LIN {X 151.175,Y 63.467,Z 53.000,A 180.000,B 0.000,C 180.000} C_DIS
LIN {X 150.850,Y 61.858,Z 53.000,A 180.000,B 0.000,C 180.000} C_DIS
LIN {X 150.811,Y 61.679,Z 53.000,A 180.000,B 0.000,C 180.000} C_DIS
LIN {X 150.487,Y 60.249,Z 53.000,A 180.000,B 0.000,C 180.000} C_DIS
LIN {X 150.447,Y 60.070,Z 53.000,A 180.000,B 0.000,C 180.000} C_DIS
LIN {X 150.402,Y 59.891,Z 53.000,A 180.000,B 0.000,C 180.000} C_DIS
LIN {X 150.042,Y 58.461,Z 53.000,A 180.000,B 0.000,C 180.000} C_DIS
LIN {X 149.995,Y 58.282,Z 53.000,A 180.000,B 0.000,C 180.000} C_DIS
LIN {X 149.600,Y 56.852,Z 53.000,A 180.000,B 0.000,C 180.000} C_DIS
LIN {X 149.550,Y 56.673,Z 53.000,A 180.000,B 0.000,C 180.000} C_DIS
LIN {X 149.497,Y 56.495,Z 53.000,A 180.000,B 0.000,C 180.000} C_DIS
LIN {X 149.065,Y 55.064,Z 53.000,A 180.000,B 0.000,C 180.000} C_DIS
LIN {X 149.008,Y 54.886,Z 53.000,A 180.000,B 0.000,C 180.000} C_DIS
LIN {X 148.540,Y 53.455,Z 53.000,A 180.000,B 0.000,C 180.000} C_DIS
LIN {X 148.480,Y 53.277,Z 53.000,A 180.000,B 0.000,C 180.000} C_DIS
LIN {X 147.974,Y 51.847,Z 53.000,A 180.000,B 0.000,C 180.000} C_DIS
LIN {X 147.911,Y 51.668,Z 53.000,A 180.000,B 0.000,C 180.000} C_DIS
LIN {X 147.846,Y 51.496,Z 53.000,A 180.000,B 0.000,C 180.000} C_DIS
LIN {X 147.299,Y 50.059,Z 53.000,A 180.000,B 0.000,C 180.000} C_DIS
LIN {X 147.227,Y 49.880,Z 53.000,A 180.000,B 0.000,C 180.000} C_DIS
LIN {X 146.645,Y 48.450,Z 53.000,A 180.000,B 0.000,C 180.000} C_DIS
LIN {X 146.595,Y 48.331,Z 53.000,A 180.000,B 0.000,C 180.000} C_DIS
LIN {X 145.947,Y 46.841,Z 53.000,A 180.000,B 0.000,C 180.000} C_DIS
LIN {X 145.880,Y 46.692,Z 53.000,A 180.000,B 0.000,C 180.000} C_DIS
LIN {X 145.203,Y 45.232,Z 53.000,A 180.000,B 0.000,C 180.000} C_DIS
LIN {X 145.164,Y 45.151,Z 53.000,A 180.000,B 0.000,C 180.000} C_DIS
LIN {X 144.449,Y 43.697,Z 53.000,A 180.000,B 0.000,C 180.000} C_DIS
LIN {X 144.413,Y 43.623,Z 53.000,A 180.000,B 0.000,C 180.000} C_DIS
LIN {X 144.320,Y 43.444,Z 53.000,A 180.000,B 0.000,C 180.000} C_DIS
LIN {X 143.668,Y 42.193,Z 53.000,A 180.000,B 0.000,C 180.000} C_DIS
LIN {X 143.574,Y 42.014,Z 53.000,A 180.000,B 0.000,C 180.000} C_DIS
LIN {X 142.785,Y 40.584,Z 53.000,A 180.000,B 0.000,C 180.000} C_DIS
LIN {X 142.683,Y 40.405,Z 53.000,A 180.000,B 0.000,C 180.000} C_DIS
LIN {X 141.947,Y 39.141,Z 53.000,A 180.000,B 0.000,C 180.000} C_DIS
LIN {X 141.849,Y 38.975,Z 53.000,A 180.000,B 0.000,C 180.000} C_DIS
LIN {X 141.768,Y 38.842,Z 53.000,A 180.000,B 0.000,C 180.000} C_DIS
LIN {X 140.971,Y 37.545,Z 53.000,A 180.000,B 0.000,C 180.000} C_DIS
LIN {X 140.874,Y 37.393,Z 53.000,A 180.000,B 0.000,C 180.000} C_DIS
LIN {X 140.047,Y 36.115,Z 53.000,A 180.000,B 0.000,C 180.000} C_DIS
LIN {X 139.980,Y 36.012,Z 53.000,A 180.000,B 0.000,C 180.000} C_DIS
LIN {X 139.928,Y 35.936,Z 53.000,A 180.000,B 0.000,C 180.000} C_DIS
LIN {X 139.076,Y 34.685,Z 53.000,A 180.000,B 0.000,C 180.000} C_DIS
LIN {X 138.953,Y 34.506,Z 53.000,A 180.000,B 0.000,C 180.000} C_DIS
LIN {X 138.014,Y 33.194,Z 53.000,A 180.000,B 0.000,C 180.000} C_DIS
LIN {X 137.927,Y 33.076,Z 53.000,A 180.000,B 0.000,C 180.000} C_DIS
LIN {X 136.941,Y 31.765,Z 53.000,A 180.000,B 0.000,C 180.000} C_DIS
LIN {X 136.848,Y 31.646,Z 53.000,A 180.000,B 0.000,C 180.000} C_DIS
LIN {X 135.861,Y 30.394,Z 53.000,A 180.000,B 0.000,C 180.000} C_DIS
LIN {X 135.714,Y 30.215,Z 53.000,A 180.000,B 0.000,C 180.000} C_DIS
LIN {X 134.796,Y 29.106,Z 53.000,A 180.000,B 0.000,C 180.000} C_DIS
LIN {X 134.677,Y 28.964,Z 53.000,A 180.000,B 0.000,C 180.000} C_DIS
LIN {X 133.590,Y 27.713,Z 53.000,A 180.000,B 0.000,C 180.000} C_DIS
LIN {X 133.544,Y 27.660,Z 53.000,A 180.000,B 0.000,C 180.000} C_DIS
LIN {X 133.430,Y 27.534,Z 53.000,A 180.000,B 0.000,C 180.000} C_DIS
LIN {X 132.453,Y 26.461,Z 53.000,A 180.000,B 0.000,C 180.000} C_DIS
LIN {X 132.293,Y 26.289,Z 53.000,A 180.000,B 0.000,C 180.000} C_DIS
LIN {X 131.220,Y 25.165,Z 53.000,A 180.000,B 0.000,C 180.000} C_DIS
LIN {X 131.090,Y 25.031,Z 53.000,A 180.000,B 0.000,C 180.000} C_DIS
LIN {X 129.969,Y 23.910,Z 53.000,A 180.000,B 0.000,C 180.000} C_DIS
LIN {X 129.835,Y 23.780,Z 53.000,A 180.000,B 0.000,C 180.000} C_DIS
LIN {X 128.711,Y 22.707,Z 53.000,A 180.000,B 0.000,C 180.000} C_DIS
LIN {X 128.539,Y 22.547,Z 53.000,A 180.000,B 0.000,C 180.000} C_DIS
LIN {X 127.466,Y 21.570,Z 53.000,A 180.000,B 0.000,C 180.000} C_DIS
LIN {X 127.340,Y 21.456,Z 53.000,A 180.000,B 0.000,C 180.000} C_DIS
LIN {X 127.287,Y 21.410,Z 53.000,A 180.000,B 0.000,C 180.000} C_DIS
LIN {X 126.036,Y 20.323,Z 53.000,A 180.000,B 0.000,C 180.000} C_DIS
LIN {X 125.894,Y 20.204,Z 53.000,A 180.000,B 0.000,C 180.000} C_DIS
LIN {X 124.785,Y 19.286,Z 53.000,A 180.000,B 0.000,C 180.000} C_DIS
LIN {X 124.606,Y 19.139,Z 53.000,A 180.000,B 0.000,C 180.000} C_DIS
LIN {X 123.354,Y 18.152,Z 53.000,A 180.000,B 0.000,C 180.000} C_DIS
LIN {X 123.235,Y 18.059,Z 53.000,A 180.000,B 0.000,C 180.000} C_DIS
LIN {X 121.924,Y 17.073,Z 53.000,A 180.000,B 0.000,C 180.000} C_DIS
LIN {X 121.806,Y 16.986,Z 53.000,A 180.000,B 0.000,C 180.000} C_DIS
LIN {X 120.494,Y 16.047,Z 53.000,A 180.000,B 0.000,C 180.000} C_DIS
LIN {X 120.315,Y 15.924,Z 53.000,A 180.000,B 0.000,C 180.000} C_DIS
LIN {X 119.064,Y 15.072,Z 53.000,A 180.000,B 0.000,C 180.000} C_DIS
LIN {X 118.988,Y 15.020,Z 53.000,A 180.000,B 0.000,C 180.000} C_DIS
LIN {X 118.885,Y 14.953,Z 53.000,A 180.000,B 0.000,C 180.000} C_DIS
LIN {X 117.607,Y 14.126,Z 53.000,A 180.000,B 0.000,C 180.000} C_DIS
LIN {X 117.455,Y 14.029,Z 53.000,A 180.000,B 0.000,C 180.000} C_DIS
LIN {X 116.158,Y 13.232,Z 53.000,A 180.000,B 0.000,C 180.000} C_DIS
LIN {X 116.025,Y 13.151,Z 53.000,A 180.000,B 0.000,C 180.000} C_DIS
LIN {X 115.859,Y 13.053,Z 53.000,A 180.000,B 0.000,C 180.000} C_DIS
LIN {X 114.595,Y 12.317,Z 53.000,A 180.000,B 0.000,C 180.000} C_DIS
LIN {X 114.416,Y 12.215,Z 53.000,A 180.000,B 0.000,C 180.000} C_DIS
LIN {X 112.986,Y 11.426,Z 53.000,A 180.000,B 0.000,C 180.000} C_DIS
LIN {X 112.807,Y 11.332,Z 53.000,A 180.000,B 0.000,C 180.000} C_DIS
LIN {X 111.556,Y 10.680,Z 53.000,A 180.000,B 0.000,C 180.000} C_DIS
LIN {X 111.377,Y 10.587,Z 53.000,A 180.000,B 0.000,C 180.000} C_DIS
LIN {X 111.303,Y 10.551,Z 53.000,A 180.000,B 0.000,C 180.000} C_DIS
LIN {X 109.849,Y 9.836,Z 53.000,A 180.000,B 0.000,C 180.000} C_DIS
LIN {X 109.768,Y 9.797,Z 53.000,A 180.000,B 0.000,C 180.000} C_DIS
LIN {X 108.308,Y 9.120,Z 53.000,A 180.000,B 0.000,C 180.000} C_DIS
LIN {X 108.159,Y 9.053,Z 53.000,A 180.000,B 0.000,C 180.000} C_DIS
LIN {X 106.669,Y 8.405,Z 53.000,A 180.000,B 0.000,C 180.000} C_DIS
LIN {X 106.550,Y 8.355,Z 53.000,A 180.000,B 0.000,C 180.000} C_DIS
LIN {X 105.120,Y 7.773,Z 53.000,A 180.000,B 0.000,C 180.000} C_DIS
LIN {X 104.941,Y 7.701,Z 53.000,A 180.000,B 0.000,C 180.000} C_DIS
LIN {X 103.504,Y 7.154,Z 53.000,A 180.000,B 0.000,C 180.000} C_DIS
LIN {X 103.332,Y 7.089,Z 53.000,A 180.000,B 0.000,C 180.000} C_DIS
LIN {X 103.153,Y 7.026,Z 53.000,A 180.000,B 0.000,C 180.000} C_DIS
LIN {X 101.723,Y 6.520,Z 53.000,A 180.000,B 0.000,C 180.000} C_DIS
LIN {X 101.545,Y 6.460,Z 53.000,A 180.000,B 0.000,C 180.000} C_DIS
LIN {X 100.114,Y 5.992,Z 53.000,A 180.000,B 0.000,C 180.000} C_DIS
LIN {X 99.936,Y 5.935,Z 53.000,A 180.000,B 0.000,C 180.000} C_DIS
LIN {X 98.505,Y 5.503,Z 53.000,A 180.000,B 0.000,C 180.000} C_DIS
LIN {X 98.327,Y 5.450,Z 53.000,A 180.000,B 0.000,C 180.000} C_DIS
LIN {X 98.148,Y 5.400,Z 53.000,A 180.000,B 0.000,C 180.000} C_DIS
LIN {X 96.718,Y 5.005,Z 53.000,A 180.000,B 0.000,C 180.000} C_DIS
LIN {X 96.539,Y 4.958,Z 53.000,A 180.000,B 0.000,C 180.000} C_DIS
LIN {X 95.109,Y 4.598,Z 53.000,A 180.000,B 0.000,C 180.000} C_DIS
LIN {X 94.930,Y 4.554,Z 53.000,A 180.000,B 0.000,C 180.000} C_DIS
LIN {X 94.751,Y 4.513,Z 53.000,A 180.000,B 0.000,C 180.000} C_DIS
LIN {X 93.321,Y 4.189,Z 53.000,A 180.000,B 0.000,C 180.000} C_DIS
LIN {X 93.142,Y 4.150,Z 53.000,A 180.000,B 0.000,C 180.000} C_DIS
LIN {X 91.533,Y 3.825,Z 53.000,A 180.000,B 0.000,C 180.000} C_DIS
LIN {X 91.355,Y 3.792,Z 53.000,A 180.000,B 0.000,C 180.000} C_DIS
LIN {X 89.925,Y 3.538,Z 53.000,A 180.000,B 0.000,C 180.000} C_DIS
LIN {X 89.746,Y 3.506,Z 53.000,A 180.000,B 0.000,C 180.000} C_DIS
LIN {X 89.567,Y 3.479,Z 53.000,A 180.000,B 0.000,C 180.000} C_DIS
LIN {X 88.137,Y 3.259,Z 53.000,A 180.000,B 0.000,C 180.000} C_DIS
LIN {X 87.958,Y 3.233,Z 53.000,A 180.000,B 0.000,C 180.000} C_DIS
LIN {X 86.349,Y 3.025,Z 53.000,A 180.000,B 0.000,C 180.000} C_DIS
LIN {X 86.170,Y 3.004,Z 53.000,A 180.000,B 0.000,C 180.000} C_DIS
LIN {X 84.561,Y 2.833,Z 53.000,A 180.000,B 0.000,C 180.000} C_DIS
LIN {X 84.383,Y 2.818,Z 53.000,A 180.000,B 0.000,C 180.000} C_DIS
LIN {X 82.952,Y 2.700,Z 53.000,A 180.000,B 0.000,C 180.000} C_DIS
LIN {X 82.774,Y 2.686,Z 53.000,A 180.000,B 0.000,C 180.000} C_DIS
LIN {X 82.761,Y 2.685,Z 53.000,A 180.000,B 0.000,C 180.000} C_DIS
LIN {X 82.595,Y 2.675,Z 53.000,A 180.000,B 0.000,C 180.000} C_DIS
LIN {X 81.165,Y 2.591,Z 53.000,A 180.000,B 0.000,C 180.000} C_DIS
LIN {X 80.986,Y 2.581,Z 53.000,A 180.000,B 0.000,C 180.000} C_DIS
LIN {X 79.377,Y 2.525,Z 53.000,A 180.000,B 0.000,C 180.000} C_DIS
LIN {X 79.198,Y 2.520,Z 53.000,A 180.000,B 0.000,C 180.000} C_DIS
LIN {X 77.589,Y 2.501,Z 53.000,A 180.000,B 0.000,C 180.000} C_DIS
LIN {X 77.411,Y 2.501,Z 53.000,A 180.000,B 0.000,C 180.000} C_DIS
LIN {X 75.802,Y 2.520,Z 53.000,A 180.000,B 0.000,C 180.000} C_DIS
LIN {X 75.623,Y 2.525,Z 53.000,A 180.000,B 0.000,C 180.000} C_DIS
LIN {X 74.014,Y 2.581,Z 53.000,A 180.000,B 0.000,C 180.000} C_DIS
LIN {X 73.835,Y 2.591,Z 53.000,A 180.000,B 0.000,C 180.000} C_DIS
LIN {X 72.405,Y 2.675,Z 53.000,A 180.000,B 0.000,C 180.000} C_DIS
LIN {X 72.239,Y 2.685,Z 53.000,A 180.000,B 0.000,C 180.000} C_DIS
LIN {X 72.226,Y 2.686,Z 53.000,A 180.000,B 0.000,C 180.000} C_DIS
LIN {X 72.048,Y 2.700,Z 53.000,A 180.000,B 0.000,C 180.000} C_DIS
LIN {X 70.617,Y 2.818,Z 53.000,A 180.000,B 0.000,C 180.000} C_DIS
LIN {X 70.439,Y 2.833,Z 53.000,A 180.000,B 0.000,C 180.000} C_DIS
LIN {X 68.830,Y 3.004,Z 53.000,A 180.000,B 0.000,C 180.000} C_DIS
LIN {X 68.651,Y 3.025,Z 53.000,A 180.000,B 0.000,C 180.000} C_DIS
LIN {X 67.042,Y 3.233,Z 53.000,A 180.000,B 0.000,C 180.000} C_DIS
LIN {X 66.863,Y 3.259,Z 53.000,A 180.000,B 0.000,C 180.000} C_DIS
LIN {X 65.433,Y 3.479,Z 53.000,A 180.000,B 0.000,C 180.000} C_DIS
LIN {X 65.254,Y 3.506,Z 53.000,A 180.000,B 0.000,C 180.000} C_DIS
LIN {X 65.075,Y 3.538,Z 53.000,A 180.000,B 0.000,C 180.000} C_DIS
LIN {X 63.645,Y 3.792,Z 53.000,A 180.000,B 0.000,C 180.000} C_DIS
LIN {X 63.467,Y 3.825,Z 53.000,A 180.000,B 0.000,C 180.000} C_DIS
LIN {X 61.858,Y 4.150,Z 53.000,A 180.000,B 0.000,C 180.000} C_DIS
LIN {X 61.679,Y 4.189,Z 53.000,A 180.000,B 0.000,C 180.000} C_DIS
LIN {X 60.249,Y 4.513,Z 53.000,A 180.000,B 0.000,C 180.000} C_DIS
LIN {X 60.070,Y 4.554,Z 53.000,A 180.000,B 0.000,C 180.000} C_DIS
LIN {X 59.891,Y 4.598,Z 53.000,A 180.000,B 0.000,C 180.000} C_DIS
LIN {X 58.461,Y 4.958,Z 53.000,A 180.000,B 0.000,C 180.000} C_DIS
LIN {X 58.282,Y 5.005,Z 53.000,A 180.000,B 0.000,C 180.000} C_DIS
LIN {X 56.852,Y 5.400,Z 53.000,A 180.000,B 0.000,C 180.000} C_DIS
LIN {X 56.673,Y 5.450,Z 53.000,A 180.000,B 0.000,C 180.000} C_DIS
LIN {X 56.495,Y 5.503,Z 53.000,A 180.000,B 0.000,C 180.000} C_DIS
LIN {X 55.064,Y 5.935,Z 53.000,A 180.000,B 0.000,C 180.000} C_DIS
LIN {X 54.886,Y 5.992,Z 53.000,A 180.000,B 0.000,C 180.000} C_DIS
LIN {X 53.455,Y 6.460,Z 53.000,A 180.000,B 0.000,C 180.000} C_DIS
LIN {X 53.277,Y 6.520,Z 53.000,A 180.000,B 0.000,C 180.000} C_DIS
LIN {X 51.847,Y 7.026,Z 53.000,A 180.000,B 0.000,C 180.000} C_DIS
LIN {X 51.668,Y 7.089,Z 53.000,A 180.000,B 0.000,C 180.000} C_DIS
LIN {X 51.496,Y 7.154,Z 53.000,A 180.000,B 0.000,C 180.000} C_DIS
LIN {X 50.059,Y 7.701,Z 53.000,A 180.000,B 0.000,C 180.000} C_DIS
LIN {X 49.880,Y 7.773,Z 53.000,A 180.000,B 0.000,C 180.000} C_DIS
LIN {X 48.450,Y 8.355,Z 53.000,A 180.000,B 0.000,C 180.000} C_DIS
LIN {X 48.331,Y 8.405,Z 53.000,A 180.000,B 0.000,C 180.000} C_DIS
LIN {X 46.841,Y 9.053,Z 53.000,A 180.000,B 0.000,C 180.000} C_DIS
LIN {X 46.692,Y 9.120,Z 53.000,A 180.000,B 0.000,C 180.000} C_DIS
LIN {X 45.232,Y 9.797,Z 53.000,A 180.000,B 0.000,C 180.000} C_DIS
LIN {X 45.151,Y 9.836,Z 53.000,A 180.000,B 0.000,C 180.000} C_DIS
LIN {X 43.697,Y 10.551,Z 53.000,A 180.000,B 0.000,C 180.000} C_DIS
LIN {X 43.623,Y 10.587,Z 53.000,A 180.000,B 0.000,C 180.000} C_DIS
LIN {X 43.444,Y 10.680,Z 53.000,A 180.000,B 0.000,C 180.000} C_DIS
LIN {X 42.193,Y 11.332,Z 53.000,A 180.000,B 0.000,C 180.000} C_DIS
LIN {X 42.014,Y 11.426,Z 53.000,A 180.000,B 0.000,C 180.000} C_DIS
LIN {X 40.584,Y 12.215,Z 53.000,A 180.000,B 0.000,C 180.000} C_DIS
LIN {X 40.405,Y 12.317,Z 53.000,A 180.000,B 0.000,C 180.000} C_DIS
LIN {X 39.141,Y 13.053,Z 53.000,A 180.000,B 0.000,C 180.000} C_DIS
LIN {X 38.975,Y 13.151,Z 53.000,A 180.000,B 0.000,C 180.000} C_DIS
LIN {X 38.842,Y 13.232,Z 53.000,A 180.000,B 0.000,C 180.000} C_DIS
LIN {X 37.545,Y 14.029,Z 53.000,A 180.000,B 0.000,C 180.000} C_DIS
LIN {X 37.393,Y 14.126,Z 53.000,A 180.000,B 0.000,C 180.000} C_DIS
LIN {X 36.115,Y 14.953,Z 53.000,A 180.000,B 0.000,C 180.000} C_DIS
LIN {X 36.012,Y 15.020,Z 53.000,A 180.000,B 0.000,C 180.000} C_DIS
LIN {X 35.936,Y 15.072,Z 53.000,A 180.000,B 0.000,C 180.000} C_DIS
LIN {X 34.685,Y 15.924,Z 53.000,A 180.000,B 0.000,C 180.000} C_DIS
LIN {X 34.506,Y 16.047,Z 53.000,A 180.000,B 0.000,C 180.000} C_DIS
LIN {X 33.194,Y 16.986,Z 53.000,A 180.000,B 0.000,C 180.000} C_DIS
LIN {X 33.076,Y 17.073,Z 53.000,A 180.000,B 0.000,C 180.000} C_DIS
LIN {X 31.765,Y 18.059,Z 53.000,A 180.000,B 0.000,C 180.000} C_DIS
LIN {X 31.646,Y 18.152,Z 53.000,A 180.000,B 0.000,C 180.000} C_DIS
LIN {X 30.394,Y 19.139,Z 53.000,A 180.000,B 0.000,C 180.000} C_DIS
LIN {X 30.215,Y 19.286,Z 53.000,A 180.000,B 0.000,C 180.000} C_DIS
LIN {X 29.106,Y 20.204,Z 53.000,A 180.000,B 0.000,C 180.000} C_DIS
LIN {X 28.964,Y 20.323,Z 53.000,A 180.000,B 0.000,C 180.000} C_DIS
LIN {X 27.713,Y 21.410,Z 53.000,A 180.000,B 0.000,C 180.000} C_DIS
LIN {X 27.660,Y 21.456,Z 53.000,A 180.000,B 0.000,C 180.000} C_DIS
LIN {X 27.534,Y 21.570,Z 53.000,A 180.000,B 0.000,C 180.000} C_DIS
LIN {X 26.461,Y 22.547,Z 53.000,A 180.000,B 0.000,C 180.000} C_DIS
LIN {X 26.289,Y 22.707,Z 53.000,A 180.000,B 0.000,C 180.000} C_DIS
LIN {X 25.165,Y 23.780,Z 53.000,A 180.000,B 0.000,C 180.000} C_DIS
LIN {X 25.031,Y 23.910,Z 53.000,A 180.000,B 0.000,C 180.000} C_DIS
LIN {X 23.910,Y 25.031,Z 53.000,A 180.000,B 0.000,C 180.000} C_DIS
LIN {X 23.780,Y 25.165,Z 53.000,A 180.000,B 0.000,C 180.000} C_DIS
LIN {X 22.707,Y 26.289,Z 53.000,A 180.000,B 0.000,C 180.000} C_DIS
LIN {X 22.547,Y 26.461,Z 53.000,A 180.000,B 0.000,C 180.000} C_DIS
LIN {X 21.570,Y 27.534,Z 53.000,A 180.000,B 0.000,C 180.000} C_DIS
LIN {X 21.456,Y 27.660,Z 53.000,A 180.000,B 0.000,C 180.000} C_DIS
LIN {X 21.410,Y 27.713,Z 53.000,A 180.000,B 0.000,C 180.000} C_DIS
LIN {X 20.323,Y 28.964,Z 53.000,A 180.000,B 0.000,C 180.000} C_DIS
LIN {X 20.204,Y 29.106,Z 53.000,A 180.000,B 0.000,C 180.000} C_DIS
LIN {X 19.286,Y 30.215,Z 53.000,A 180.000,B 0.000,C 180.000} C_DIS
LIN {X 19.139,Y 30.394,Z 53.000,A 180.000,B 0.000,C 180.000} C_DIS
LIN {X 18.152,Y 31.646,Z 53.000,A 180.000,B 0.000,C 180.000} C_DIS
LIN {X 18.059,Y 31.765,Z 53.000,A 180.000,B 0.000,C 180.000} C_DIS
LIN {X 17.073,Y 33.076,Z 53.000,A 180.000,B 0.000,C 180.000} C_DIS
LIN {X 16.986,Y 33.194,Z 53.000,A 180.000,B 0.000,C 180.000} C_DIS
LIN {X 16.047,Y 34.506,Z 53.000,A 180.000,B 0.000,C 180.000} C_DIS
LIN {X 15.924,Y 34.685,Z 53.000,A 180.000,B 0.000,C 180.000} C_DIS
LIN {X 15.072,Y 35.936,Z 53.000,A 180.000,B 0.000,C 180.000} C_DIS
LIN {X 15.020,Y 36.012,Z 53.000,A 180.000,B 0.000,C 180.000} C_DIS
LIN {X 14.953,Y 36.115,Z 53.000,A 180.000,B 0.000,C 180.000} C_DIS
LIN {X 14.126,Y 37.393,Z 53.000,A 180.000,B 0.000,C 180.000} C_DIS
LIN {X 14.029,Y 37.545,Z 53.000,A 180.000,B 0.000,C 180.000} C_DIS
LIN {X 13.232,Y 38.842,Z 53.000,A 180.000,B 0.000,C 180.000} C_DIS
LIN {X 13.151,Y 38.975,Z 53.000,A 180.000,B 0.000,C 180.000} C_DIS
LIN {X 13.053,Y 39.141,Z 53.000,A 180.000,B 0.000,C 180.000} C_DIS
LIN {X 12.317,Y 40.405,Z 53.000,A 180.000,B 0.000,C 180.000} C_DIS
LIN {X 12.215,Y 40.584,Z 53.000,A 180.000,B 0.000,C 180.000} C_DIS
LIN {X 11.426,Y 42.014,Z 53.000,A 180.000,B 0.000,C 180.000} C_DIS
LIN {X 11.332,Y 42.193,Z 53.000,A 180.000,B 0.000,C 180.000} C_DIS
LIN {X 10.680,Y 43.444,Z 53.000,A 180.000,B 0.000,C 180.000} C_DIS
LIN {X 10.587,Y 43.623,Z 53.000,A 180.000,B 0.000,C 180.000} C_DIS
LIN {X 10.551,Y 43.697,Z 53.000,A 180.000,B 0.000,C 180.000} C_DIS
LIN {X 9.836,Y 45.151,Z 53.000,A 180.000,B 0.000,C 180.000} C_DIS
LIN {X 9.797,Y 45.232,Z 53.000,A 180.000,B 0.000,C 180.000} C_DIS
LIN {X 9.120,Y 46.692,Z 53.000,A 180.000,B 0.000,C 180.000} C_DIS
LIN {X 9.053,Y 46.841,Z 53.000,A 180.000,B 0.000,C 180.000} C_DIS
LIN {X 8.405,Y 48.331,Z 53.000,A 180.000,B 0.000,C 180.000} C_DIS
LIN {X 8.355,Y 48.450,Z 53.000,A 180.000,B 0.000,C 180.000} C_DIS
LIN {X 7.773,Y 49.880,Z 53.000,A 180.000,B 0.000,C 180.000} C_DIS
LIN {X 7.701,Y 50.059,Z 53.000,A 180.000,B 0.000,C 180.000} C_DIS
LIN {X 7.154,Y 51.496,Z 53.000,A 180.000,B 0.000,C 180.000} C_DIS
LIN {X 7.089,Y 51.668,Z 53.000,A 180.000,B 0.000,C 180.000} C_DIS
LIN {X 7.026,Y 51.847,Z 53.000,A 180.000,B 0.000,C 180.000} C_DIS
LIN {X 6.520,Y 53.277,Z 53.000,A 180.000,B 0.000,C 180.000} C_DIS
LIN {X 6.460,Y 53.455,Z 53.000,A 180.000,B 0.000,C 180.000} C_DIS
LIN {X 5.992,Y 54.886,Z 53.000,A 180.000,B 0.000,C 180.000} C_DIS
LIN {X 5.935,Y 55.064,Z 53.000,A 180.000,B 0.000,C 180.000} C_DIS
LIN {X 5.503,Y 56.495,Z 53.000,A 180.000,B 0.000,C 180.000} C_DIS
LIN {X 5.450,Y 56.673,Z 53.000,A 180.000,B 0.000,C 180.000} C_DIS
LIN {X 5.400,Y 56.852,Z 53.000,A 180.000,B 0.000,C 180.000} C_DIS
LIN {X 5.005,Y 58.282,Z 53.000,A 180.000,B 0.000,C 180.000} C_DIS
LIN {X 4.958,Y 58.461,Z 53.000,A 180.000,B 0.000,C 180.000} C_DIS
LIN {X 4.598,Y 59.891,Z 53.000,A 180.000,B 0.000,C 180.000} C_DIS
LIN {X 4.554,Y 60.070,Z 53.000,A 180.000,B 0.000,C 180.000} C_DIS
LIN {X 4.513,Y 60.249,Z 53.000,A 180.000,B 0.000,C 180.000} C_DIS
LIN {X 4.189,Y 61.679,Z 53.000,A 180.000,B 0.000,C 180.000} C_DIS
LIN {X 4.150,Y 61.858,Z 53.000,A 180.000,B 0.000,C 180.000} C_DIS
LIN {X 3.825,Y 63.467,Z 53.000,A 180.000,B 0.000,C 180.000} C_DIS
LIN {X 3.792,Y 63.645,Z 53.000,A 180.000,B 0.000,C 180.000} C_DIS
LIN {X 3.538,Y 65.075,Z 53.000,A 180.000,B 0.000,C 180.000} C_DIS
LIN {X 3.506,Y 65.254,Z 53.000,A 180.000,B 0.000,C 180.000} C_DIS
LIN {X 3.479,Y 65.433,Z 53.000,A 180.000,B 0.000,C 180.000} C_DIS
LIN {X 3.259,Y 66.863,Z 53.000,A 180.000,B 0.000,C 180.000} C_DIS
LIN {X 3.233,Y 67.042,Z 53.000,A 180.000,B 0.000,C 180.000} C_DIS
LIN {X 3.025,Y 68.651,Z 53.000,A 180.000,B 0.000,C 180.000} C_DIS
LIN {X 3.004,Y 68.830,Z 53.000,A 180.000,B 0.000,C 180.000} C_DIS
LIN {X 2.833,Y 70.439,Z 53.000,A 180.000,B 0.000,C 180.000} C_DIS
LIN {X 2.818,Y 70.617,Z 53.000,A 180.000,B 0.000,C 180.000} C_DIS
LIN {X 2.700,Y 72.048,Z 53.000,A 180.000,B 0.000,C 180.000} C_DIS
LIN {X 2.686,Y 72.226,Z 53.000,A 180.000,B 0.000,C 180.000} C_DIS
LIN {X 2.685,Y 72.239,Z 53.000,A 180.000,B 0.000,C 180.000} C_DIS
LIN {X 2.675,Y 72.405,Z 53.000,A 180.000,B 0.000,C 180.000} C_DIS
LIN {X 2.591,Y 73.835,Z 53.000,A 180.000,B 0.000,C 180.000} C_DIS
LIN {X 2.581,Y 74.014,Z 53.000,A 180.000,B 0.000,C 180.000} C_DIS
LIN {X 2.525,Y 75.623,Z 53.000,A 180.000,B 0.000,C 180.000} C_DIS
LIN {X 2.520,Y 75.802,Z 53.000,A 180.000,B 0.000,C 180.000} C_DIS
LIN {X 2.506,Y 76.973,Z 53.000,A 180.000,B 0.000,C 180.000} C_DIS
LIN {X 2.501,Y 77.411,Z 53.000,A 180.000,B 0.000,C 180.000} C_DIS
LIN {X 2.501,Y 77.589,Z 53.000,A 180.000,B 0.000,C 180.000} C_DIS
LIN {X 2.520,Y 79.198,Z 53.000,A 180.000,B 0.000,C 180.000} C_DIS
LIN {X 2.525,Y 79.377,Z 53.000,A 180.000,B 0.000,C 180.000} C_DIS
LIN {X 2.581,Y 80.986,Z 53.000,A 180.000,B 0.000,C 180.000} C_DIS
LIN {X 2.591,Y 81.165,Z 53.000,A 180.000,B 0.000,C 180.000} C_DIS
LIN {X 2.675,Y 82.595,Z 53.000,A 180.000,B 0.000,C 180.000} C_DIS
LIN {X 2.685,Y 82.761,Z 53.000,A 180.000,B 0.000,C 180.000} C_DIS
LIN {X 2.686,Y 82.774,Z 53.000,A 180.000,B 0.000,C 180.000} C_DIS
LIN {X 2.700,Y 82.952,Z 53.000,A 180.000,B 0.000,C 180.000} C_DIS
LIN {X 2.818,Y 84.383,Z 53.000,A 180.000,B 0.000,C 180.000} C_DIS
LIN {X 2.833,Y 84.561,Z 53.000,A 180.000,B 0.000,C 180.000} C_DIS
LIN {X 3.004,Y 86.170,Z 53.000,A 180.000,B 0.000,C 180.000} C_DIS
LIN {X 3.025,Y 86.349,Z 53.000,A 180.000,B 0.000,C 180.000} C_DIS
LIN {X 3.233,Y 87.958,Z 53.000,A 180.000,B 0.000,C 180.000} C_DIS
LIN {X 3.259,Y 88.137,Z 53.000,A 180.000,B 0.000,C 180.000} C_DIS
LIN {X 3.479,Y 89.567,Z 53.000,A 180.000,B 0.000,C 180.000} C_DIS
LIN {X 3.506,Y 89.746,Z 53.000,A 180.000,B 0.000,C 180.000} C_DIS
LIN {X 3.538,Y 89.925,Z 53.000,A 180.000,B 0.000,C 180.000} C_DIS
LIN {X 3.792,Y 91.355,Z 53.000,A 180.000,B 0.000,C 180.000} C_DIS
LIN {X 3.825,Y 91.533,Z 53.000,A 180.000,B 0.000,C 180.000} C_DIS
LIN {X 4.150,Y 93.142,Z 53.000,A 180.000,B 0.000,C 180.000} C_DIS
LIN {X 4.189,Y 93.321,Z 53.000,A 180.000,B 0.000,C 180.000} C_DIS
LIN {X 4.513,Y 94.751,Z 53.000,A 180.000,B 0.000,C 180.000} C_DIS
LIN {X 4.554,Y 94.930,Z 53.000,A 180.000,B 0.000,C 180.000} C_DIS
LIN {X 4.598,Y 95.109,Z 53.000,A 180.000,B 0.000,C 180.000} C_DIS
LIN {X 4.958,Y 96.539,Z 53.000,A 180.000,B 0.000,C 180.000} C_DIS
LIN {X 5.005,Y 96.718,Z 53.000,A 180.000,B 0.000,C 180.000} C_DIS
LIN {X 5.400,Y 98.148,Z 53.000,A 180.000,B 0.000,C 180.000} C_DIS
LIN {X 5.450,Y 98.327,Z 53.000,A 180.000,B 0.000,C 180.000} C_DIS
LIN {X 5.503,Y 98.505,Z 53.000,A 180.000,B 0.000,C 180.000} C_DIS
LIN {X 5.935,Y 99.936,Z 53.000,A 180.000,B 0.000,C 180.000} C_DIS
LIN {X 5.992,Y 100.114,Z 53.000,A 180.000,B 0.000,C 180.000} C_DIS
LIN {X 6.460,Y 101.545,Z 53.000,A 180.000,B 0.000,C 180.000} C_DIS
LIN {X 6.520,Y 101.723,Z 53.000,A 180.000,B 0.000,C 180.000} C_DIS
LIN {X 7.026,Y 103.153,Z 53.000,A 180.000,B 0.000,C 180.000} C_DIS
LIN {X 7.089,Y 103.332,Z 53.000,A 180.000,B 0.000,C 180.000} C_DIS
LIN {X 7.154,Y 103.504,Z 53.000,A 180.000,B 0.000,C 180.000} C_DIS
LIN {X 7.701,Y 104.941,Z 53.000,A 180.000,B 0.000,C 180.000} C_DIS
LIN {X 7.773,Y 105.120,Z 53.000,A 180.000,B 0.000,C 180.000} C_DIS
LIN {X 8.355,Y 106.550,Z 53.000,A 180.000,B 0.000,C 180.000} C_DIS
LIN {X 8.405,Y 106.669,Z 53.000,A 180.000,B 0.000,C 180.000} C_DIS
LIN {X 9.053,Y 108.159,Z 53.000,A 180.000,B 0.000,C 180.000} C_DIS
LIN {X 9.120,Y 108.308,Z 53.000,A 180.000,B 0.000,C 180.000} C_DIS
LIN {X 9.797,Y 109.768,Z 53.000,A 180.000,B 0.000,C 180.000} C_DIS
LIN {X 9.836,Y 109.849,Z 53.000,A 180.000,B 0.000,C 180.000} C_DIS
LIN {X 10.551,Y 111.303,Z 53.000,A 180.000,B 0.000,C 180.000} C_DIS
LIN {X 10.587,Y 111.377,Z 53.000,A 180.000,B 0.000,C 180.000} C_DIS
LIN {X 10.680,Y 111.556,Z 53.000,A 180.000,B 0.000,C 180.000} C_DIS
LIN {X 11.332,Y 112.807,Z 53.000,A 180.000,B 0.000,C 180.000} C_DIS
LIN {X 11.426,Y 112.986,Z 53.000,A 180.000,B 0.000,C 180.000} C_DIS
LIN {X 12.215,Y 114.416,Z 53.000,A 180.000,B 0.000,C 180.000} C_DIS
LIN {X 12.317,Y 114.595,Z 53.000,A 180.000,B 0.000,C 180.000} C_DIS
LIN {X 13.053,Y 115.859,Z 53.000,A 180.000,B 0.000,C 180.000} C_DIS
LIN {X 13.151,Y 116.025,Z 53.000,A 180.000,B 0.000,C 180.000} C_DIS
LIN {X 13.232,Y 116.158,Z 53.000,A 180.000,B 0.000,C 180.000} C_DIS
LIN {X 14.029,Y 117.455,Z 53.000,A 180.000,B 0.000,C 180.000} C_DIS
LIN {X 14.126,Y 117.607,Z 53.000,A 180.000,B 0.000,C 180.000} C_DIS
LIN {X 14.953,Y 118.885,Z 53.000,A 180.000,B 0.000,C 180.000} C_DIS
LIN {X 15.020,Y 118.988,Z 53.000,A 180.000,B 0.000,C 180.000} C_DIS
LIN {X 15.072,Y 119.064,Z 53.000,A 180.000,B 0.000,C 180.000} C_DIS
LIN {X 15.924,Y 120.315,Z 53.000,A 180.000,B 0.000,C 180.000} C_DIS
LIN {X 16.047,Y 120.494,Z 53.000,A 180.000,B 0.000,C 180.000} C_DIS
LIN {X 16.986,Y 121.806,Z 53.000,A 180.000,B 0.000,C 180.000} C_DIS
LIN {X 17.073,Y 121.924,Z 53.000,A 180.000,B 0.000,C 180.000} C_DIS
LIN {X 18.059,Y 123.235,Z 53.000,A 180.000,B 0.000,C 180.000} C_DIS
LIN {X 18.152,Y 123.354,Z 53.000,A 180.000,B 0.000,C 180.000} C_DIS
LIN {X 19.139,Y 124.606,Z 53.000,A 180.000,B 0.000,C 180.000} C_DIS
LIN {X 19.286,Y 124.785,Z 53.000,A 180.000,B 0.000,C 180.000} C_DIS
LIN {X 20.204,Y 125.894,Z 53.000,A 180.000,B 0.000,C 180.000} C_DIS
LIN {X 20.323,Y 126.036,Z 53.000,A 180.000,B 0.000,C 180.000} C_DIS
LIN {X 21.410,Y 127.287,Z 53.000,A 180.000,B 0.000,C 180.000} C_DIS
LIN {X 21.456,Y 127.340,Z 53.000,A 180.000,B 0.000,C 180.000} C_DIS
LIN {X 21.570,Y 127.466,Z 53.000,A 180.000,B 0.000,C 180.000} C_DIS
LIN {X 22.547,Y 128.539,Z 53.000,A 180.000,B 0.000,C 180.000} C_DIS
LIN {X 22.707,Y 128.711,Z 53.000,A 180.000,B 0.000,C 180.000} C_DIS
LIN {X 23.780,Y 129.835,Z 53.000,A 180.000,B 0.000,C 180.000} C_DIS
LIN {X 23.910,Y 129.969,Z 53.000,A 180.000,B 0.000,C 180.000} C_DIS
LIN {X 25.031,Y 131.090,Z 53.000,A 180.000,B 0.000,C 180.000} C_DIS
LIN {X 25.165,Y 131.220,Z 53.000,A 180.000,B 0.000,C 180.000} C_DIS
LIN {X 26.289,Y 132.293,Z 53.000,A 180.000,B 0.000,C 180.000} C_DIS
LIN {X 26.461,Y 132.453,Z 53.000,A 180.000,B 0.000,C 180.000} C_DIS
LIN {X 27.534,Y 133.430,Z 53.000,A 180.000,B 0.000,C 180.000} C_DIS
LIN {X 27.660,Y 133.544,Z 53.000,A 180.000,B 0.000,C 180.000} C_DIS
LIN {X 27.713,Y 133.590,Z 53.000,A 180.000,B 0.000,C 180.000} C_DIS
LIN {X 28.964,Y 134.677,Z 53.000,A 180.000,B 0.000,C 180.000} C_DIS
LIN {X 29.106,Y 134.796,Z 53.000,A 180.000,B 0.000,C 180.000} C_DIS
LIN {X 30.215,Y 135.714,Z 53.000,A 180.000,B 0.000,C 180.000} C_DIS
LIN {X 30.394,Y 135.861,Z 53.000,A 180.000,B 0.000,C 180.000} C_DIS
LIN {X 31.646,Y 136.848,Z 53.000,A 180.000,B 0.000,C 180.000} C_DIS
LIN {X 31.765,Y 136.941,Z 53.000,A 180.000,B 0.000,C 180.000} C_DIS
LIN {X 33.076,Y 137.927,Z 53.000,A 180.000,B 0.000,C 180.000} C_DIS
LIN {X 33.194,Y 138.014,Z 53.000,A 180.000,B 0.000,C 180.000} C_DIS
LIN {X 34.506,Y 138.953,Z 53.000,A 180.000,B 0.000,C 180.000} C_DIS
LIN {X 34.685,Y 139.076,Z 53.000,A 180.000,B 0.000,C 180.000} C_DIS
LIN {X 35.936,Y 139.928,Z 53.000,A 180.000,B 0.000,C 180.000} C_DIS
LIN {X 36.012,Y 139.980,Z 53.000,A 180.000,B 0.000,C 180.000} C_DIS
LIN {X 36.115,Y 140.047,Z 53.000,A 180.000,B 0.000,C 180.000} C_DIS
LIN {X 37.393,Y 140.874,Z 53.000,A 180.000,B 0.000,C 180.000} C_DIS
LIN {X 37.545,Y 140.971,Z 53.000,A 180.000,B 0.000,C 180.000} C_DIS
LIN {X 38.842,Y 141.768,Z 53.000,A 180.000,B 0.000,C 180.000} C_DIS
LIN {X 38.975,Y 141.849,Z 53.000,A 180.000,B 0.000,C 180.000} C_DIS
LIN {X 39.141,Y 141.947,Z 53.000,A 180.000,B 0.000,C 180.000} C_DIS
LIN {X 40.405,Y 142.683,Z 53.000,A 180.000,B 0.000,C 180.000} C_DIS
LIN {X 40.584,Y 142.785,Z 53.000,A 180.000,B 0.000,C 180.000} C_DIS
LIN {X 42.014,Y 143.574,Z 53.000,A 180.000,B 0.000,C 180.000} C_DIS
LIN {X 42.193,Y 143.668,Z 53.000,A 180.000,B 0.000,C 180.000} C_DIS
LIN {X 43.444,Y 144.320,Z 53.000,A 180.000,B 0.000,C 180.000} C_DIS
LIN {X 43.623,Y 144.413,Z 53.000,A 180.000,B 0.000,C 180.000} C_DIS
LIN {X 43.697,Y 144.449,Z 53.000,A 180.000,B 0.000,C 180.000} C_DIS
LIN {X 45.151,Y 145.164,Z 53.000,A 180.000,B 0.000,C 180.000} C_DIS
LIN {X 45.232,Y 145.203,Z 53.000,A 180.000,B 0.000,C 180.000} C_DIS
LIN {X 46.692,Y 145.880,Z 53.000,A 180.000,B 0.000,C 180.000} C_DIS
LIN {X 46.841,Y 145.947,Z 53.000,A 180.000,B 0.000,C 180.000} C_DIS
LIN {X 48.331,Y 146.595,Z 53.000,A 180.000,B 0.000,C 180.000} C_DIS
LIN {X 48.450,Y 146.645,Z 53.000,A 180.000,B 0.000,C 180.000} C_DIS
LIN {X 49.880,Y 147.227,Z 53.000,A 180.000,B 0.000,C 180.000} C_DIS
LIN {X 50.059,Y 147.299,Z 53.000,A 180.000,B 0.000,C 180.000} C_DIS
LIN {X 51.496,Y 147.846,Z 53.000,A 180.000,B 0.000,C 180.000} C_DIS
LIN {X 51.668,Y 147.911,Z 53.000,A 180.000,B 0.000,C 180.000} C_DIS
LIN {X 51.847,Y 147.974,Z 53.000,A 180.000,B 0.000,C 180.000} C_DIS
LIN {X 53.277,Y 148.480,Z 53.000,A 180.000,B 0.000,C 180.000} C_DIS
LIN {X 53.455,Y 148.540,Z 53.000,A 180.000,B 0.000,C 180.000} C_DIS
LIN {X 54.290,Y 148.813,Z 53.000,A 180.000,B 0.000,C 180.000} C_DIS
LIN {X 54.886,Y 149.008,Z 53.000,A 180.000,B 0.000,C 180.000} C_DIS
LIN {X 55.064,Y 149.065,Z 53.000,A 180.000,B 0.000,C 180.000} C_DIS
LIN {X 56.495,Y 149.497,Z 53.000,A 180.000,B 0.000,C 180.000} C_DIS
LIN {X 56.673,Y 149.550,Z 53.000,A 180.000,B 0.000,C 180.000} C_DIS
LIN {X 56.852,Y 149.600,Z 53.000,A 180.000,B 0.000,C 180.000} C_DIS
LIN {X 58.282,Y 149.995,Z 53.000,A 180.000,B 0.000,C 180.000} C_DIS
LIN {X 58.461,Y 150.042,Z 53.000,A 180.000,B 0.000,C 180.000} C_DIS
LIN {X 59.891,Y 150.402,Z 53.000,A 180.000,B 0.000,C 180.000} C_DIS
LIN {X 60.070,Y 150.447,Z 53.000,A 180.000,B 0.000,C 180.000} C_DIS
LIN {X 60.249,Y 150.487,Z 53.000,A 180.000,B 0.000,C 180.000} C_DIS
LIN {X 61.679,Y 150.811,Z 53.000,A 180.000,B 0.000,C 180.000} C_DIS
LIN {X 61.858,Y 150.850,Z 53.000,A 180.000,B 0.000,C 180.000} C_DIS
LIN {X 63.467,Y 151.175,Z 53.000,A 180.000,B 0.000,C 180.000} C_DIS
LIN {X 63.645,Y 151.208,Z 53.000,A 180.000,B 0.000,C 180.000} C_DIS
LIN {X 65.075,Y 151.462,Z 53.000,A 180.000,B 0.000,C 180.000} C_DIS
LIN {X 65.254,Y 151.494,Z 53.000,A 180.000,B 0.000,C 180.000} C_DIS
LIN {X 65.433,Y 151.521,Z 53.000,A 180.000,B 0.000,C 180.000} C_DIS
LIN {X 66.863,Y 151.741,Z 53.000,A 180.000,B 0.000,C 180.000} C_DIS
LIN {X 67.042,Y 151.767,Z 53.000,A 180.000,B 0.000,C 180.000} C_DIS
LIN {X 68.651,Y 151.975,Z 53.000,A 180.000,B 0.000,C 180.000} C_DIS
LIN {X 68.830,Y 151.996,Z 53.000,A 180.000,B 0.000,C 180.000} C_DIS
LIN {X 70.439,Y 152.167,Z 53.000,A 180.000,B 0.000,C 180.000} C_DIS
LIN {X 70.617,Y 152.182,Z 53.000,A 180.000,B 0.000,C 180.000} C_DIS
LIN {X 72.048,Y 152.300,Z 53.000,A 180.000,B 0.000,C 180.000} C_DIS
LIN {X 72.226,Y 152.314,Z 53.000,A 180.000,B 0.000,C 180.000} C_DIS
LIN {X 72.239,Y 152.315,Z 53.000,A 180.000,B 0.000,C 180.000} C_DIS
LIN {X 72.405,Y 152.325,Z 53.000,A 180.000,B 0.000,C 180.000} C_DIS
LIN {X 73.835,Y 152.409,Z 53.000,A 180.000,B 0.000,C 180.000} C_DIS
LIN {X 74.014,Y 152.419,Z 53.000,A 180.000,B 0.000,C 180.000} C_DIS
LIN {X 75.623,Y 152.475,Z 53.000,A 180.000,B 0.000,C 180.000} C_DIS
LIN {X 75.802,Y 152.480,Z 53.000,A 180.000,B 0.000,C 180.000} C_DIS
LIN {X 77.411,Y 152.499,Z 53.000,A 180.000,B 0.000,C 180.000} C_DIS
LIN {X 77.589,Y 152.499,Z 53.000,A 180.000,B 0.000,C 180.000} C_DIS
LIN {X 79.198,Y 152.480,Z 53.000,A 180.000,B 0.000,C 180.000} C_DIS
LIN {X 79.377,Y 152.475,Z 53.000,A 180.000,B 0.000,C 180.000} C_DIS
LIN {X 80.986,Y 152.419,Z 53.000,A 180.000,B 0.000,C 180.000} C_DIS
LIN {X 81.165,Y 152.409,Z 53.000,A 180.000,B 0.000,C 180.000} C_DIS
LIN {X 82.595,Y 152.325,Z 53.000,A 180.000,B 0.000,C 180.000} C_DIS
LIN {X 82.761,Y 152.315,Z 53.000,A 180.000,B 0.000,C 180.000} C_DIS
LIN {X 82.774,Y 152.314,Z 53.000,A 180.000,B 0.000,C 180.000} C_DIS
LIN {X 82.952,Y 152.300,Z 53.000,A 180.000,B 0.000,C 180.000} C_DIS
LIN {X 84.383,Y 152.182,Z 53.000,A 180.000,B 0.000,C 180.000} C_DIS
LIN {X 84.561,Y 152.167,Z 53.000,A 180.000,B 0.000,C 180.000} C_DIS
LIN {X 86.170,Y 151.996,Z 53.000,A 180.000,B 0.000,C 180.000} C_DIS
LIN {X 86.349,Y 151.975,Z 53.000,A 180.000,B 0.000,C 180.000} C_DIS
LIN {X 87.958,Y 151.767,Z 53.000,A 180.000,B 0.000,C 180.000} C_DIS
LIN {X 88.137,Y 151.741,Z 53.000,A 180.000,B 0.000,C 180.000} C_DIS
LIN {X 89.567,Y 151.521,Z 53.000,A 180.000,B 0.000,C 180.000} C_DIS
LIN {X 89.746,Y 151.494,Z 53.000,A 180.000,B 0.000,C 180.000} C_DIS
LIN {X 89.925,Y 151.462,Z 53.000,A 180.000,B 0.000,C 180.000} C_DIS
LIN {X 91.355,Y 151.208,Z 53.000,A 180.000,B 0.000,C 180.000} C_DIS
LIN {X 91.533,Y 151.175,Z 53.000,A 180.000,B 0.000,C 180.000} C_DIS
LIN {X 93.142,Y 150.850,Z 53.000,A 180.000,B 0.000,C 180.000} C_DIS
LIN {X 93.321,Y 150.811,Z 53.000,A 180.000,B 0.000,C 180.000} C_DIS
LIN {X 94.751,Y 150.487,Z 53.000,A 180.000,B 0.000,C 180.000} C_DIS
LIN {X 94.930,Y 150.447,Z 53.000,A 180.000,B 0.000,C 180.000} C_DIS
LIN {X 95.109,Y 150.402,Z 53.000,A 180.000,B 0.000,C 180.000} C_DIS
LIN {X 96.539,Y 150.042,Z 53.000,A 180.000,B 0.000,C 180.000} C_DIS
LIN {X 96.718,Y 149.995,Z 53.000,A 180.000,B 0.000,C 180.000} C_DIS
LIN {X 98.148,Y 149.600,Z 53.000,A 180.000,B 0.000,C 180.000} C_DIS
LIN {X 98.327,Y 149.550,Z 53.000,A 180.000,B 0.000,C 180.000} C_DIS
LIN {X 98.505,Y 149.497,Z 53.000,A 180.000,B 0.000,C 180.000} C_DIS
LIN {X 99.936,Y 149.065,Z 53.000,A 180.000,B 0.000,C 180.000} C_DIS
LIN {X 100.114,Y 149.008,Z 53.000,A 180.000,B 0.000,C 180.000} C_DIS
LIN {X 101.545,Y 148.540,Z 53.000,A 180.000,B 0.000,C 180.000} C_DIS
LIN {X 101.723,Y 148.480,Z 53.000,A 180.000,B 0.000,C 180.000} C_DIS
LIN {X 103.153,Y 147.974,Z 53.000,A 180.000,B 0.000,C 180.000} C_DIS
LIN {X 103.332,Y 147.911,Z 53.000,A 180.000,B 0.000,C 180.000} C_DIS
LIN {X 103.504,Y 147.846,Z 53.000,A 180.000,B 0.000,C 180.000} C_DIS
LIN {X 104.941,Y 147.299,Z 53.000,A 180.000,B 0.000,C 180.000} C_DIS
LIN {X 105.120,Y 147.227,Z 53.000,A 180.000,B 0.000,C 180.000} C_DIS
LIN {X 106.550,Y 146.645,Z 53.000,A 180.000,B 0.000,C 180.000} C_DIS
LIN {X 106.669,Y 146.595,Z 53.000,A 180.000,B 0.000,C 180.000} C_DIS
LIN {X 108.159,Y 145.947,Z 53.000,A 180.000,B 0.000,C 180.000} C_DIS
LIN {X 108.308,Y 145.880,Z 53.000,A 180.000,B 0.000,C 180.000} C_DIS
LIN {X 109.768,Y 145.203,Z 53.000,A 180.000,B 0.000,C 180.000} C_DIS
LIN {X 109.849,Y 145.164,Z 53.000,A 180.000,B 0.000,C 180.000} C_DIS
LIN {X 111.303,Y 144.449,Z 53.000,A 180.000,B 0.000,C 180.000} C_DIS
LIN {X 111.377,Y 144.413,Z 53.000,A 180.000,B 0.000,C 180.000} C_DIS
LIN {X 111.556,Y 144.320,Z 53.000,A 180.000,B 0.000,C 180.000} C_DIS
LIN {X 112.807,Y 143.668,Z 53.000,A 180.000,B 0.000,C 180.000} C_DIS
LIN {X 112.986,Y 143.574,Z 53.000,A 180.000,B 0.000,C 180.000} C_DIS
LIN {X 114.416,Y 142.785,Z 53.000,A 180.000,B 0.000,C 180.000} C_DIS
LIN {X 114.595,Y 142.683,Z 53.000,A 180.000,B 0.000,C 180.000} C_DIS
LIN {X 115.859,Y 141.947,Z 53.000,A 180.000,B 0.000,C 180.000} C_DIS
LIN {X 116.025,Y 141.849,Z 53.000,A 180.000,B 0.000,C 180.000} C_DIS
LIN {X 116.158,Y 141.768,Z 53.000,A 180.000,B 0.000,C 180.000} C_DIS
LIN {X 117.455,Y 140.971,Z 53.000,A 180.000,B 0.000,C 180.000} C_DIS
LIN {X 117.607,Y 140.874,Z 53.000,A 180.000,B 0.000,C 180.000} C_DIS
LIN {X 118.885,Y 140.047,Z 53.000,A 180.000,B 0.000,C 180.000} C_DIS
LIN {X 118.988,Y 139.980,Z 53.000,A 180.000,B 0.000,C 180.000} C_DIS
LIN {X 119.064,Y 139.928,Z 53.000,A 180.000,B 0.000,C 180.000} C_DIS
LIN {X 120.315,Y 139.076,Z 53.000,A 180.000,B 0.000,C 180.000} C_DIS
LIN {X 120.494,Y 138.953,Z 53.000,A 180.000,B 0.000,C 180.000} C_DIS
LIN {X 121.806,Y 138.014,Z 53.000,A 180.000,B 0.000,C 180.000} C_DIS
LIN {X 121.924,Y 137.927,Z 53.000,A 180.000,B 0.000,C 180.000} C_DIS
LIN {X 122.641,Y 137.388,Z 53.000,A 180.000,B 0.000,C 180.000} C_DIS
LIN {X 123.235,Y 136.941,Z 53.000,A 180.000,B 0.000,C 180.000} C_DIS
LIN {X 123.354,Y 136.848,Z 53.000,A 180.000,B 0.000,C 180.000} C_DIS
LIN {X 124.606,Y 135.861,Z 53.000,A 180.000,B 0.000,C 180.000} C_DIS
LIN {X 124.785,Y 135.714,Z 53.000,A 180.000,B 0.000,C 180.000} C_DIS
LIN {X 125.894,Y 134.796,Z 53.000,A 180.000,B 0.000,C 180.000} C_DIS
LIN {X 126.036,Y 134.677,Z 53.000,A 180.000,B 0.000,C 180.000} C_DIS
LIN {X 127.287,Y 133.590,Z 53.000,A 180.000,B 0.000,C 180.000} C_DIS
LIN {X 127.340,Y 133.544,Z 53.000,A 180.000,B 0.000,C 180.000} C_DIS
LIN {X 127.466,Y 133.430,Z 53.000,A 180.000,B 0.000,C 180.000} C_DIS
LIN {X 128.539,Y 132.453,Z 53.000,A 180.000,B 0.000,C 180.000} C_DIS
LIN {X 128.711,Y 132.293,Z 53.000,A 180.000,B 0.000,C 180.000} C_DIS
LIN {X 129.835,Y 131.220,Z 53.000,A 180.000,B 0.000,C 180.000} C_DIS
LIN {X 129.969,Y 131.090,Z 53.000,A 180.000,B 0.000,C 180.000} C_DIS
LIN {X 131.090,Y 129.969,Z 53.000,A 180.000,B 0.000,C 180.000} C_DIS
LIN {X 131.220,Y 129.835,Z 53.000,A 180.000,B 0.000,C 180.000} C_DIS
LIN {X 132.293,Y 128.711,Z 53.000,A 180.000,B 0.000,C 180.000} C_DIS
LIN {X 132.453,Y 128.539,Z 53.000,A 180.000,B 0.000,C 180.000} C_DIS
LIN {X 133.430,Y 127.466,Z 53.000,A 180.000,B 0.000,C 180.000} C_DIS
LIN {X 133.544,Y 127.340,Z 53.000,A 180.000,B 0.000,C 180.000} C_DIS
LIN {X 133.590,Y 127.287,Z 53.000,A 180.000,B 0.000,C 180.000} C_DIS
LIN {X 134.677,Y 126.036,Z 53.000,A 180.000,B 0.000,C 180.000} C_DIS
LIN {X 134.796,Y 125.894,Z 53.000,A 180.000,B 0.000,C 180.000} C_DIS
LIN {X 135.714,Y 124.785,Z 53.000,A 180.000,B 0.000,C 180.000} C_DIS
LIN {X 135.861,Y 124.606,Z 53.000,A 180.000,B 0.000,C 180.000} C_DIS
LIN {X 136.848,Y 123.354,Z 53.000,A 180.000,B 0.000,C 180.000} C_DIS
LIN {X 136.941,Y 123.235,Z 53.000,A 180.000,B 0.000,C 180.000} C_DIS
LIN {X 137.927,Y 121.924,Z 53.000,A 180.000,B 0.000,C 180.000} C_DIS
LIN {X 138.014,Y 121.806,Z 53.000,A 180.000,B 0.000,C 180.000} C_DIS
LIN {X 138.953,Y 120.494,Z 53.000,A 180.000,B 0.000,C 180.000} C_DIS
LIN {X 139.076,Y 120.315,Z 53.000,A 180.000,B 0.000,C 180.000} C_DIS
LIN {X 139.928,Y 119.064,Z 53.000,A 180.000,B 0.000,C 180.000} C_DIS
LIN {X 139.980,Y 118.988,Z 53.000,A 180.000,B 0.000,C 180.000} C_DIS
LIN {X 140.047,Y 118.885,Z 53.000,A 180.000,B 0.000,C 180.000} C_DIS
LIN {X 140.874,Y 117.607,Z 53.000,A 180.000,B 0.000,C 180.000} C_DIS
LIN {X 140.971,Y 117.455,Z 53.000,A 180.000,B 0.000,C 180.000} C_DIS
LIN {X 141.768,Y 116.158,Z 53.000,A 180.000,B 0.000,C 180.000} C_DIS
LIN {X 141.849,Y 116.025,Z 53.000,A 180.000,B 0.000,C 180.000} C_DIS
LIN {X 141.947,Y 115.859,Z 53.000,A 180.000,B 0.000,C 180.000} C_DIS
LIN {X 142.683,Y 114.595,Z 53.000,A 180.000,B 0.000,C 180.000} C_DIS
LIN {X 142.785,Y 114.416,Z 53.000,A 180.000,B 0.000,C 180.000} C_DIS
LIN {X 143.574,Y 112.986,Z 53.000,A 180.000,B 0.000,C 180.000} C_DIS
LIN {X 143.668,Y 112.807,Z 53.000,A 180.000,B 0.000,C 180.000} C_DIS
LIN {X 144.320,Y 111.556,Z 53.000,A 180.000,B 0.000,C 180.000} C_DIS
LIN {X 144.413,Y 111.377,Z 53.000,A 180.000,B 0.000,C 180.000} C_DIS
LIN {X 144.449,Y 111.303,Z 53.000,A 180.000,B 0.000,C 180.000} C_DIS
LIN {X 145.164,Y 109.849,Z 53.000,A 180.000,B 0.000,C 180.000} C_DIS
LIN {X 145.203,Y 109.768,Z 53.000,A 180.000,B 0.000,C 180.000} C_DIS
LIN {X 145.656,Y 108.791,Z 53.000,A 180.000,B 0.000,C 180.000} C_DIS
; Link Move Starts
LIN {X 145.788,Y 108.505,Z 53.000,A 180.000,B 0.000,C 180.000} C_DIS
LIN {X 145.920,Y 108.219,Z 52.999,A 180.000,B 0.000,C 180.000} C_DIS
LIN {X 146.046,Y 107.930,Z 52.998,A 180.000,B 0.000,C 180.000} C_DIS
LIN {X 146.172,Y 107.642,Z 52.996,A 180.000,B 0.000,C 180.000} C_DIS
LIN {X 146.297,Y 107.353,Z 52.994,A 180.000,B 0.000,C 180.000} C_DIS
LIN {X 146.423,Y 107.064,Z 52.991,A 180.000,B 0.000,C 180.000} C_DIS
LIN {X 146.549,Y 106.775,Z 52.988,A 180.000,B 0.000,C 180.000} C_DIS
LIN {X 146.671,Y 106.485,Z 52.985,A 180.000,B 0.000,C 180.000} C_DIS
LIN {X 146.790,Y 106.193,Z 52.981,A 180.000,B 0.000,C 180.000} C_DIS
LIN {X 146.909,Y 105.902,Z 52.977,A 180.000,B 0.000,C 180.000} C_DIS
LIN {X 147.028,Y 105.610,Z 52.972,A 180.000,B 0.000,C 180.000} C_DIS
LIN {X 147.087,Y 105.464,Z 52.969,A 180.000,B 0.000,C 180.000} C_DIS
LIN {X 147.147,Y 105.318,Z 52.967,A 180.000,B 0.000,C 180.000} C_DIS
LIN {X 147.206,Y 105.172,Z 52.964,A 180.000,B 0.000,C 180.000} C_DIS
LIN {X 147.266,Y 105.026,Z 52.961,A 180.000,B 0.000,C 180.000} C_DIS
LIN {X 147.323,Y 104.880,Z 52.959,A 180.000,B 0.000,C 180.000} C_DIS
LIN {X 147.379,Y 104.732,Z 52.956,A 180.000,B 0.000,C 180.000} C_DIS
LIN {X 147.435,Y 104.585,Z 52.952,A 180.000,B 0.000,C 180.000} C_DIS
LIN {X 147.491,Y 104.438,Z 52.949,A 180.000,B 0.000,C 180.000} C_DIS
LIN {X 147.547,Y 104.291,Z 52.946,A 180.000,B 0.000,C 180.000} C_DIS
LIN {X 147.603,Y 104.144,Z 52.943,A 180.000,B 0.000,C 180.000} C_DIS
LIN {X 147.659,Y 103.996,Z 52.939,A 180.000,B 0.000,C 180.000} C_DIS
LIN {X 147.715,Y 103.849,Z 52.936,A 180.000,B 0.000,C 180.000} C_DIS
LIN {X 147.771,Y 103.702,Z 52.932,A 180.000,B 0.000,C 180.000} C_DIS
LIN {X 147.827,Y 103.555,Z 52.928,A 180.000,B 0.000,C 180.000} C_DIS
LIN {X 147.883,Y 103.407,Z 52.925,A 180.000,B 0.000,C 180.000} C_DIS
LIN {X 147.937,Y 103.260,Z 52.921,A 180.000,B 0.000,C 180.000} C_DIS
LIN {X 147.989,Y 103.111,Z 52.917,A 180.000,B 0.000,C 180.000} C_DIS
LIN {X 148.042,Y 102.963,Z 52.913,A 180.000,B 0.000,C 180.000} C_DIS
LIN {X 148.094,Y 102.814,Z 52.909,A 180.000,B 0.000,C 180.000} C_DIS
LIN {X 148.147,Y 102.666,Z 52.905,A 180.000,B 0.000,C 180.000} C_DIS
LIN {X 148.199,Y 102.517,Z 52.900,A 180.000,B 0.000,C 180.000} C_DIS
LIN {X 148.252,Y 102.369,Z 52.896,A 180.000,B 0.000,C 180.000} C_DIS
LIN {X 148.304,Y 102.220,Z 52.892,A 180.000,B 0.000,C 180.000} C_DIS
LIN {X 148.357,Y 102.072,Z 52.887,A 180.000,B 0.000,C 180.000} C_DIS
LIN {X 148.409,Y 101.923,Z 52.883,A 180.000,B 0.000,C 180.000} C_DIS
LIN {X 148.462,Y 101.775,Z 52.878,A 180.000,B 0.000,C 180.000} C_DIS
LIN {X 148.513,Y 101.626,Z 52.873,A 180.000,B 0.000,C 180.000} C_DIS
LIN {X 148.562,Y 101.476,Z 52.869,A 180.000,B 0.000,C 180.000} C_DIS
LIN {X 148.611,Y 101.326,Z 52.864,A 180.000,B 0.000,C 180.000} C_DIS
LIN {X 148.660,Y 101.177,Z 52.859,A 180.000,B 0.000,C 180.000} C_DIS
LIN {X 148.709,Y 101.027,Z 52.854,A 180.000,B 0.000,C 180.000} C_DIS
LIN {X 148.734,Y 100.952,Z 52.851,A 180.000,B 0.000,C 180.000} C_DIS
LIN {X 148.758,Y 100.877,Z 52.849,A 180.000,B 0.000,C 180.000} C_DIS
LIN {X 148.783,Y 100.803,Z 52.846,A 180.000,B 0.000,C 180.000} C_DIS
LIN {X 148.807,Y 100.728,Z 52.844,A 180.000,B 0.000,C 180.000} C_DIS
LIN {X 148.832,Y 100.653,Z 52.841,A 180.000,B 0.000,C 180.000} C_DIS
LIN {X 148.856,Y 100.578,Z 52.839,A 180.000,B 0.000,C 180.000} C_DIS
LIN {X 148.881,Y 100.503,Z 52.836,A 180.000,B 0.000,C 180.000} C_DIS
LIN {X 148.930,Y 100.354,Z 52.831,A 180.000,B 0.000,C 180.000} C_DIS
LIN {X 148.979,Y 100.204,Z 52.825,A 180.000,B 0.000,C 180.000} C_DIS
LIN {X 149.028,Y 100.054,Z 52.820,A 180.000,B 0.000,C 180.000} C_DIS
LIN {X 149.052,Y 99.979,Z 52.817,A 180.000,B 0.000,C 180.000} C_DIS
LIN {X 149.097,Y 99.828,Z 52.812,A 180.000,B 0.000,C 180.000} C_DIS
LIN {X 149.188,Y 99.527,Z 52.801,A 180.000,B 0.000,C 180.000} C_DIS
LIN {X 149.257,Y 99.301,Z 52.793,A 180.000,B 0.000,C 180.000} C_DIS
LIN {X 149.302,Y 99.150,Z 52.787,A 180.000,B 0.000,C 180.000} C_DIS
LIN {X 149.325,Y 99.074,Z 52.785,A 180.000,B 0.000,C 180.000} C_DIS
LIN {X 149.370,Y 98.924,Z 52.779,A 180.000,B 0.000,C 180.000} C_DIS
LIN {X 149.439,Y 98.698,Z 52.771,A 180.000,B 0.000,C 180.000} C_DIS
LIN {X 149.484,Y 98.547,Z 52.765,A 180.000,B 0.000,C 180.000} C_DIS
LIN {X 149.507,Y 98.471,Z 52.763,A 180.000,B 0.000,C 180.000} C_DIS
LIN {X 149.530,Y 98.396,Z 52.760,A 180.000,B 0.000,C 180.000} C_DIS
LIN {X 149.552,Y 98.320,Z 52.757,A 180.000,B 0.000,C 180.000} C_DIS
LIN {X 149.573,Y 98.245,Z 52.754,A 180.000,B 0.000,C 180.000} C_DIS
LIN {X 149.594,Y 98.169,Z 52.752,A 180.000,B 0.000,C 180.000} C_DIS
LIN {X 149.636,Y 98.017,Z 52.746,A 180.000,B 0.000,C 180.000} C_DIS
LIN {X 149.699,Y 97.789,Z 52.738,A 180.000,B 0.000,C 180.000} C_DIS
LIN {X 149.741,Y 97.637,Z 52.732,A 180.000,B 0.000,C 180.000} C_DIS
LIN {X 149.762,Y 97.561,Z 52.730,A 180.000,B 0.000,C 180.000} C_DIS
LIN {X 149.804,Y 97.410,Z 52.724,A 180.000,B 0.000,C 180.000} C_DIS
LIN {X 149.930,Y 96.954,Z 52.708,A 180.000,B 0.000,C 180.000} C_DIS
LIN {X 149.972,Y 96.802,Z 52.702,A 180.000,B 0.000,C 180.000} C_DIS
LIN {X 150.014,Y 96.651,Z 52.697,A 180.000,B 0.000,C 180.000} C_DIS
LIN {X 150.033,Y 96.574,Z 52.694,A 180.000,B 0.000,C 180.000} C_DIS
LIN {X 150.072,Y 96.422,Z 52.688,A 180.000,B 0.000,C 180.000} C_DIS
LIN {X 150.091,Y 96.345,Z 52.686,A 180.000,B 0.000,C 180.000} C_DIS
LIN {X 150.129,Y 96.193,Z 52.680,A 180.000,B 0.000,C 180.000} C_DIS
LIN {X 150.245,Y 95.734,Z 52.664,A 180.000,B 0.000,C 180.000} C_DIS
LIN {X 150.302,Y 95.505,Z 52.655,A 180.000,B 0.000,C 180.000} C_DIS
LIN {X 150.340,Y 95.352,Z 52.650,A 180.000,B 0.000,C 180.000} C_DIS
LIN {X 150.436,Y 94.970,Z 52.636,A 180.000,B 0.000,C 180.000} C_DIS
LIN {X 150.455,Y 94.894,Z 52.633,A 180.000,B 0.000,C 180.000} C_DIS
LIN {X 150.490,Y 94.740,Z 52.628,A 180.000,B 0.000,C 180.000} C_DIS
LIN {X 150.594,Y 94.280,Z 52.611,A 180.000,B 0.000,C 180.000} C_DIS
LIN {X 150.629,Y 94.126,Z 52.606,A 180.000,B 0.000,C 180.000} C_DIS
LIN {X 150.803,Y 93.358,Z 52.578,A 180.000,B 0.000,C 180.000} C_DIS
LIN {X 150.820,Y 93.281,Z 52.576,A 180.000,B 0.000,C 180.000} C_DIS
LIN {X 150.837,Y 93.204,Z 52.573,A 180.000,B 0.000,C 180.000} C_DIS
LIN {X 150.853,Y 93.127,Z 52.570,A 180.000,B 0.000,C 180.000} C_DIS
LIN {X 151.134,Y 91.738,Z 52.521,A 180.000,B 0.000,C 180.000} C_DIS
LIN {X 151.181,Y 91.506,Z 52.512,A 180.000,B 0.000,C 180.000} C_DIS
LIN {X 151.195,Y 91.429,Z 52.510,A 180.000,B 0.000,C 180.000} C_DIS
LIN {X 151.484,Y 89.800,Z 52.452,A 180.000,B 0.000,C 180.000} C_DIS
LIN {X 151.497,Y 89.723,Z 52.449,A 180.000,B 0.000,C 180.000} C_DIS
LIN {X 151.724,Y 88.244,Z 52.397,A 180.000,B 0.000,C 180.000} C_DIS
LIN {X 151.748,Y 88.088,Z 52.391,A 180.000,B 0.000,C 180.000} C_DIS
LIN {X 151.760,Y 88.010,Z 52.389,A 180.000,B 0.000,C 180.000} C_DIS
LIN {X 151.770,Y 87.932,Z 52.386,A 180.000,B 0.000,C 180.000} C_DIS
LIN {X 151.831,Y 87.464,Z 52.369,A 180.000,B 0.000,C 180.000} C_DIS
LIN {X 151.851,Y 87.307,Z 52.364,A 180.000,B 0.000,C 180.000} C_DIS
LIN {X 151.912,Y 86.839,Z 52.347,A 180.000,B 0.000,C 180.000} C_DIS
LIN {X 151.932,Y 86.683,Z 52.342,A 180.000,B 0.000,C 180.000} C_DIS
LIN {X 151.973,Y 86.370,Z 52.331,A 180.000,B 0.000,C 180.000} C_DIS
LIN {X 151.983,Y 86.292,Z 52.328,A 180.000,B 0.000,C 180.000} C_DIS
LIN {X 151.992,Y 86.214,Z 52.325,A 180.000,B 0.000,C 180.000} C_DIS
LIN {X 152.000,Y 86.136,Z 52.323,A 180.000,B 0.000,C 180.000} C_DIS
LIN {X 152.016,Y 85.979,Z 52.317,A 180.000,B 0.000,C 180.000} C_DIS
LIN {X 152.066,Y 85.509,Z 52.301,A 180.000,B 0.000,C 180.000} C_DIS
LIN {X 152.083,Y 85.352,Z 52.295,A 180.000,B 0.000,C 180.000} C_DIS
LIN {X 152.133,Y 84.883,Z 52.279,A 180.000,B 0.000,C 180.000} C_DIS
LIN {X 152.149,Y 84.726,Z 52.273,A 180.000,B 0.000,C 180.000} C_DIS
LIN {X 152.166,Y 84.569,Z 52.268,A 180.000,B 0.000,C 180.000} C_DIS
LIN {X 152.173,Y 84.491,Z 52.265,A 180.000,B 0.000,C 180.000} C_DIS
LIN {X 152.186,Y 84.334,Z 52.259,A 180.000,B 0.000,C 180.000} C_DIS
LIN {X 152.193,Y 84.255,Z 52.257,A 180.000,B 0.000,C 180.000} C_DIS
LIN {X 152.206,Y 84.098,Z 52.251,A 180.000,B 0.000,C 180.000} C_DIS
LIN {X 152.225,Y 83.863,Z 52.243,A 180.000,B 0.000,C 180.000} C_DIS
LIN {X 152.238,Y 83.706,Z 52.237,A 180.000,B 0.000,C 180.000} C_DIS
LIN {X 152.244,Y 83.628,Z 52.235,A 180.000,B 0.000,C 180.000} C_DIS
LIN {X 152.257,Y 83.471,Z 52.229,A 180.000,B 0.000,C 180.000} C_DIS
LIN {X 152.277,Y 83.235,Z 52.221,A 180.000,B 0.000,C 180.000} C_DIS
LIN {X 152.289,Y 83.078,Z 52.215,A 180.000,B 0.000,C 180.000} C_DIS
LIN {X 152.296,Y 83.000,Z 52.213,A 180.000,B 0.000,C 180.000} C_DIS
LIN {X 152.309,Y 82.843,Z 52.207,A 180.000,B 0.000,C 180.000} C_DIS
LIN {X 152.315,Y 82.764,Z 52.204,A 180.000,B 0.000,C 180.000} C_DIS
LIN {X 152.320,Y 82.686,Z 52.202,A 180.000,B 0.000,C 180.000} C_DIS
LIN {X 152.329,Y 82.528,Z 52.196,A 180.000,B 0.000,C 180.000} C_DIS
LIN {X 152.338,Y 82.371,Z 52.191,A 180.000,B 0.000,C 180.000} C_DIS
LIN {X 152.347,Y 82.214,Z 52.185,A 180.000,B 0.000,C 180.000} C_DIS
LIN {X 152.357,Y 82.057,Z 52.180,A 180.000,B 0.000,C 180.000} C_DIS
LIN {X 152.366,Y 81.899,Z 52.174,A 180.000,B 0.000,C 180.000} C_DIS
LIN {X 152.375,Y 81.742,Z 52.169,A 180.000,B 0.000,C 180.000} C_DIS
LIN {X 152.384,Y 81.585,Z 52.164,A 180.000,B 0.000,C 180.000} C_DIS
LIN {X 152.389,Y 81.506,Z 52.161,A 180.000,B 0.000,C 180.000} C_DIS
LIN {X 152.394,Y 81.428,Z 52.159,A 180.000,B 0.000,C 180.000} C_DIS
LIN {X 152.398,Y 81.349,Z 52.156,A 180.000,B 0.000,C 180.000} C_DIS
LIN {X 152.403,Y 81.271,Z 52.154,A 180.000,B 0.000,C 180.000} C_DIS
LIN {X 152.407,Y 81.192,Z 52.151,A 180.000,B 0.000,C 180.000} C_DIS
LIN {X 152.412,Y 81.113,Z 52.148,A 180.000,B 0.000,C 180.000} C_DIS
LIN {X 152.420,Y 80.956,Z 52.143,A 180.000,B 0.000,C 180.000} C_DIS
LIN {X 152.425,Y 80.799,Z 52.139,A 180.000,B 0.000,C 180.000} C_DIS
LIN {X 152.431,Y 80.641,Z 52.134,A 180.000,B 0.000,C 180.000} C_DIS
LIN {X 152.436,Y 80.484,Z 52.129,A 180.000,B 0.000,C 180.000} C_DIS
LIN {X 152.442,Y 80.326,Z 52.124,A 180.000,B 0.000,C 180.000} C_DIS
LIN {X 152.448,Y 80.169,Z 52.120,A 180.000,B 0.000,C 180.000} C_DIS
LIN {X 152.453,Y 80.012,Z 52.115,A 180.000,B 0.000,C 180.000} C_DIS
LIN {X 152.459,Y 79.854,Z 52.110,A 180.000,B 0.000,C 180.000} C_DIS
LIN {X 152.464,Y 79.697,Z 52.106,A 180.000,B 0.000,C 180.000} C_DIS
LIN {X 152.470,Y 79.539,Z 52.102,A 180.000,B 0.000,C 180.000} C_DIS
LIN {X 152.475,Y 79.382,Z 52.097,A 180.000,B 0.000,C 180.000} C_DIS
LIN {X 152.480,Y 79.225,Z 52.093,A 180.000,B 0.000,C 180.000} C_DIS
LIN {X 152.482,Y 79.067,Z 52.089,A 180.000,B 0.000,C 180.000} C_DIS
LIN {X 152.484,Y 78.910,Z 52.085,A 180.000,B 0.000,C 180.000} C_DIS
LIN {X 152.485,Y 78.752,Z 52.081,A 180.000,B 0.000,C 180.000} C_DIS
LIN {X 152.487,Y 78.595,Z 52.077,A 180.000,B 0.000,C 180.000} C_DIS
LIN {X 152.489,Y 78.437,Z 52.073,A 180.000,B 0.000,C 180.000} C_DIS
LIN {X 152.491,Y 78.280,Z 52.070,A 180.000,B 0.000,C 180.000} C_DIS
LIN {X 152.493,Y 78.122,Z 52.066,A 180.000,B 0.000,C 180.000} C_DIS
LIN {X 152.495,Y 77.965,Z 52.062,A 180.000,B 0.000,C 180.000} C_DIS
LIN {X 152.497,Y 77.807,Z 52.059,A 180.000,B 0.000,C 180.000} C_DIS
LIN {X 152.498,Y 77.650,Z 52.056,A 180.000,B 0.000,C 180.000} C_DIS
LIN {X 152.500,Y 77.492,Z 52.052,A 180.000,B 0.000,C 180.000} C_DIS
LIN {X 152.498,Y 77.335,Z 52.049,A 180.000,B 0.000,C 180.000} C_DIS
LIN {X 152.496,Y 77.177,Z 52.046,A 180.000,B 0.000,C 180.000} C_DIS
LIN {X 152.495,Y 77.020,Z 52.043,A 180.000,B 0.000,C 180.000} C_DIS
LIN {X 152.493,Y 76.862,Z 52.040,A 180.000,B 0.000,C 180.000} C_DIS
LIN {X 152.491,Y 76.705,Z 52.037,A 180.000,B 0.000,C 180.000} C_DIS
LIN {X 152.489,Y 76.547,Z 52.034,A 180.000,B 0.000,C 180.000} C_DIS
LIN {X 152.487,Y 76.390,Z 52.032,A 180.000,B 0.000,C 180.000} C_DIS
LIN {X 152.485,Y 76.232,Z 52.029,A 180.000,B 0.000,C 180.000} C_DIS
LIN {X 152.483,Y 76.075,Z 52.027,A 180.000,B 0.000,C 180.000} C_DIS
LIN {X 152.480,Y 75.760,Z 52.022,A 180.000,B 0.000,C 180.000} C_DIS
LIN {X 152.469,Y 75.445,Z 52.018,A 180.000,B 0.000,C 180.000} C_DIS
LIN {X 152.458,Y 75.130,Z 52.014,A 180.000,B 0.000,C 180.000} C_DIS
LIN {X 152.447,Y 74.815,Z 52.011,A 180.000,B 0.000,C 180.000} C_DIS
LIN {X 152.436,Y 74.501,Z 52.008,A 180.000,B 0.000,C 180.000} C_DIS
LIN {X 152.425,Y 74.186,Z 52.005,A 180.000,B 0.000,C 180.000} C_DIS
LIN {X 152.411,Y 73.871,Z 52.003,A 180.000,B 0.000,C 180.000} C_DIS
LIN {X 152.393,Y 73.557,Z 52.002,A 180.000,B 0.000,C 180.000} C_DIS
LIN {X 152.374,Y 73.242,Z 52.001,A 180.000,B 0.000,C 180.000} C_DIS
LIN {X 152.356,Y 72.928,Z 52.000,A 180.000,B 0.000,C 180.000} C_DIS
LIN {X 152.342,Y 72.697,Z 52.000,A 180.000,B 0.000,C 180.000} C_DIS
; Cutting Move Starts
LIN {X 152.325,Y 72.405,Z 52.000,A 180.000,B 0.000,C 180.000} C_DIS
LIN {X 152.315,Y 72.239,Z 52.000,A 180.000,B 0.000,C 180.000} C_DIS
LIN {X 152.314,Y 72.226,Z 52.000,A 180.000,B 0.000,C 180.000} C_DIS
LIN {X 152.300,Y 72.048,Z 52.000,A 180.000,B 0.000,C 180.000} C_DIS
LIN {X 152.182,Y 70.617,Z 52.000,A 180.000,B 0.000,C 180.000} C_DIS
LIN {X 152.167,Y 70.439,Z 52.000,A 180.000,B 0.000,C 180.000} C_DIS
LIN {X 151.996,Y 68.830,Z 52.000,A 180.000,B 0.000,C 180.000} C_DIS
LIN {X 151.975,Y 68.651,Z 52.000,A 180.000,B 0.000,C 180.000} C_DIS
LIN {X 151.767,Y 67.042,Z 52.000,A 180.000,B 0.000,C 180.000} C_DIS
LIN {X 151.741,Y 66.863,Z 52.000,A 180.000,B 0.000,C 180.000} C_DIS
LIN {X 151.521,Y 65.433,Z 52.000,A 180.000,B 0.000,C 180.000} C_DIS
LIN {X 151.494,Y 65.254,Z 52.000,A 180.000,B 0.000,C 180.000} C_DIS
LIN {X 151.462,Y 65.075,Z 52.000,A 180.000,B 0.000,C 180.000} C_DIS
LIN {X 151.208,Y 63.645,Z 52.000,A 180.000,B 0.000,C 180.000} C_DIS
LIN {X 151.175,Y 63.467,Z 52.000,A 180.000,B 0.000,C 180.000} C_DIS
LIN {X 150.850,Y 61.858,Z 52.000,A 180.000,B 0.000,C 180.000} C_DIS
LIN {X 150.811,Y 61.679,Z 52.000,A 180.000,B 0.000,C 180.000} C_DIS
LIN {X 150.487,Y 60.249,Z 52.000,A 180.000,B 0.000,C 180.000} C_DIS
LIN {X 150.447,Y 60.070,Z 52.000,A 180.000,B 0.000,C 180.000} C_DIS
LIN {X 150.402,Y 59.891,Z 52.000,A 180.000,B 0.000,C 180.000} C_DIS
LIN {X 150.042,Y 58.461,Z 52.000,A 180.000,B 0.000,C 180.000} C_DIS
LIN {X 149.995,Y 58.282,Z 52.000,A 180.000,B 0.000,C 180.000} C_DIS
LIN {X 149.600,Y 56.852,Z 52.000,A 180.000,B 0.000,C 180.000} C_DIS
LIN {X 149.550,Y 56.673,Z 52.000,A 180.000,B 0.000,C 180.000} C_DIS
LIN {X 149.497,Y 56.495,Z 52.000,A 180.000,B 0.000,C 180.000} C_DIS
LIN {X 149.065,Y 55.064,Z 52.000,A 180.000,B 0.000,C 180.000} C_DIS
LIN {X 149.008,Y 54.886,Z 52.000,A 180.000,B 0.000,C 180.000} C_DIS
LIN {X 148.540,Y 53.455,Z 52.000,A 180.000,B 0.000,C 180.000} C_DIS
LIN {X 148.480,Y 53.277,Z 52.000,A 180.000,B 0.000,C 180.000} C_DIS
LIN {X 147.974,Y 51.847,Z 52.000,A 180.000,B 0.000,C 180.000} C_DIS
LIN {X 147.911,Y 51.668,Z 52.000,A 180.000,B 0.000,C 180.000} C_DIS
LIN {X 147.846,Y 51.496,Z 52.000,A 180.000,B 0.000,C 180.000} C_DIS
LIN {X 147.299,Y 50.059,Z 52.000,A 180.000,B 0.000,C 180.000} C_DIS
LIN {X 147.227,Y 49.880,Z 52.000,A 180.000,B 0.000,C 180.000} C_DIS
LIN {X 146.645,Y 48.450,Z 52.000,A 180.000,B 0.000,C 180.000} C_DIS
LIN {X 146.595,Y 48.331,Z 52.000,A 180.000,B 0.000,C 180.000} C_DIS
LIN {X 145.947,Y 46.841,Z 52.000,A 180.000,B 0.000,C 180.000} C_DIS
LIN {X 145.880,Y 46.692,Z 52.000,A 180.000,B 0.000,C 180.000} C_DIS
LIN {X 145.203,Y 45.232,Z 52.000,A 180.000,B 0.000,C 180.000} C_DIS
LIN {X 145.164,Y 45.151,Z 52.000,A 180.000,B 0.000,C 180.000} C_DIS
LIN {X 144.449,Y 43.697,Z 52.000,A 180.000,B 0.000,C 180.000} C_DIS
LIN {X 144.413,Y 43.623,Z 52.000,A 180.000,B 0.000,C 180.000} C_DIS
LIN {X 144.320,Y 43.444,Z 52.000,A 180.000,B 0.000,C 180.000} C_DIS
LIN {X 143.668,Y 42.193,Z 52.000,A 180.000,B 0.000,C 180.000} C_DIS
LIN {X 143.574,Y 42.014,Z 52.000,A 180.000,B 0.000,C 180.000} C_DIS
LIN {X 142.785,Y 40.584,Z 52.000,A 180.000,B 0.000,C 180.000} C_DIS
LIN {X 142.683,Y 40.405,Z 52.000,A 180.000,B 0.000,C 180.000} C_DIS
LIN {X 141.947,Y 39.141,Z 52.000,A 180.000,B 0.000,C 180.000} C_DIS
LIN {X 141.849,Y 38.975,Z 52.000,A 180.000,B 0.000,C 180.000} C_DIS
LIN {X 141.768,Y 38.842,Z 52.000,A 180.000,B 0.000,C 180.000} C_DIS
LIN {X 140.971,Y 37.545,Z 52.000,A 180.000,B 0.000,C 180.000} C_DIS
LIN {X 140.874,Y 37.393,Z 52.000,A 180.000,B 0.000,C 180.000} C_DIS
LIN {X 140.047,Y 36.115,Z 52.000,A 180.000,B 0.000,C 180.000} C_DIS
LIN {X 139.980,Y 36.012,Z 52.000,A 180.000,B 0.000,C 180.000} C_DIS
LIN {X 139.928,Y 35.936,Z 52.000,A 180.000,B 0.000,C 180.000} C_DIS
LIN {X 139.076,Y 34.685,Z 52.000,A 180.000,B 0.000,C 180.000} C_DIS
LIN {X 138.953,Y 34.506,Z 52.000,A 180.000,B 0.000,C 180.000} C_DIS
LIN {X 138.014,Y 33.194,Z 52.000,A 180.000,B 0.000,C 180.000} C_DIS
LIN {X 137.927,Y 33.076,Z 52.000,A 180.000,B 0.000,C 180.000} C_DIS
LIN {X 136.941,Y 31.765,Z 52.000,A 180.000,B 0.000,C 180.000} C_DIS
LIN {X 136.848,Y 31.646,Z 52.000,A 180.000,B 0.000,C 180.000} C_DIS
LIN {X 135.861,Y 30.394,Z 52.000,A 180.000,B 0.000,C 180.000} C_DIS
LIN {X 135.714,Y 30.215,Z 52.000,A 180.000,B 0.000,C 180.000} C_DIS
LIN {X 134.796,Y 29.106,Z 52.000,A 180.000,B 0.000,C 180.000} C_DIS
LIN {X 134.677,Y 28.964,Z 52.000,A 180.000,B 0.000,C 180.000} C_DIS
LIN {X 133.590,Y 27.713,Z 52.000,A 180.000,B 0.000,C 180.000} C_DIS
LIN {X 133.544,Y 27.660,Z 52.000,A 180.000,B 0.000,C 180.000} C_DIS
LIN {X 133.430,Y 27.534,Z 52.000,A 180.000,B 0.000,C 180.000} C_DIS
LIN {X 132.453,Y 26.461,Z 52.000,A 180.000,B 0.000,C 180.000} C_DIS
LIN {X 132.293,Y 26.289,Z 52.000,A 180.000,B 0.000,C 180.000} C_DIS
LIN {X 131.220,Y 25.165,Z 52.000,A 180.000,B 0.000,C 180.000} C_DIS
LIN {X 131.090,Y 25.031,Z 52.000,A 180.000,B 0.000,C 180.000} C_DIS
LIN {X 129.969,Y 23.910,Z 52.000,A 180.000,B 0.000,C 180.000} C_DIS
LIN {X 129.835,Y 23.780,Z 52.000,A 180.000,B 0.000,C 180.000} C_DIS
LIN {X 128.711,Y 22.707,Z 52.000,A 180.000,B 0.000,C 180.000} C_DIS
LIN {X 128.539,Y 22.547,Z 52.000,A 180.000,B 0.000,C 180.000} C_DIS
LIN {X 127.466,Y 21.570,Z 52.000,A 180.000,B 0.000,C 180.000} C_DIS
LIN {X 127.340,Y 21.456,Z 52.000,A 180.000,B 0.000,C 180.000} C_DIS
LIN {X 127.287,Y 21.410,Z 52.000,A 180.000,B 0.000,C 180.000} C_DIS
LIN {X 126.036,Y 20.323,Z 52.000,A 180.000,B 0.000,C 180.000} C_DIS
LIN {X 125.894,Y 20.204,Z 52.000,A 180.000,B 0.000,C 180.000} C_DIS
LIN {X 124.785,Y 19.286,Z 52.000,A 180.000,B 0.000,C 180.000} C_DIS
LIN {X 124.606,Y 19.139,Z 52.000,A 180.000,B 0.000,C 180.000} C_DIS
LIN {X 123.354,Y 18.152,Z 52.000,A 180.000,B 0.000,C 180.000} C_DIS
LIN {X 123.235,Y 18.059,Z 52.000,A 180.000,B 0.000,C 180.000} C_DIS
LIN {X 121.924,Y 17.073,Z 52.000,A 180.000,B 0.000,C 180.000} C_DIS
LIN {X 121.806,Y 16.986,Z 52.000,A 180.000,B 0.000,C 180.000} C_DIS
LIN {X 120.494,Y 16.047,Z 52.000,A 180.000,B 0.000,C 180.000} C_DIS
LIN {X 120.315,Y 15.924,Z 52.000,A 180.000,B 0.000,C 180.000} C_DIS
LIN {X 119.064,Y 15.072,Z 52.000,A 180.000,B 0.000,C 180.000} C_DIS
LIN {X 118.988,Y 15.020,Z 52.000,A 180.000,B 0.000,C 180.000} C_DIS
LIN {X 118.885,Y 14.953,Z 52.000,A 180.000,B 0.000,C 180.000} C_DIS
LIN {X 117.607,Y 14.126,Z 52.000,A 180.000,B 0.000,C 180.000} C_DIS
LIN {X 117.455,Y 14.029,Z 52.000,A 180.000,B 0.000,C 180.000} C_DIS
LIN {X 116.158,Y 13.232,Z 52.000,A 180.000,B 0.000,C 180.000} C_DIS
LIN {X 116.025,Y 13.151,Z 52.000,A 180.000,B 0.000,C 180.000} C_DIS
LIN {X 115.859,Y 13.053,Z 52.000,A 180.000,B 0.000,C 180.000} C_DIS
LIN {X 114.595,Y 12.317,Z 52.000,A 180.000,B 0.000,C 180.000} C_DIS
LIN {X 114.416,Y 12.215,Z 52.000,A 180.000,B 0.000,C 180.000} C_DIS
LIN {X 112.986,Y 11.426,Z 52.000,A 180.000,B 0.000,C 180.000} C_DIS
LIN {X 112.807,Y 11.332,Z 52.000,A 180.000,B 0.000,C 180.000} C_DIS
LIN {X 111.556,Y 10.680,Z 52.000,A 180.000,B 0.000,C 180.000} C_DIS
LIN {X 111.377,Y 10.587,Z 52.000,A 180.000,B 0.000,C 180.000} C_DIS
LIN {X 111.303,Y 10.551,Z 52.000,A 180.000,B 0.000,C 180.000} C_DIS
LIN {X 109.849,Y 9.836,Z 52.000,A 180.000,B 0.000,C 180.000} C_DIS
LIN {X 109.768,Y 9.797,Z 52.000,A 180.000,B 0.000,C 180.000} C_DIS
LIN {X 108.308,Y 9.120,Z 52.000,A 180.000,B 0.000,C 180.000} C_DIS
LIN {X 108.159,Y 9.053,Z 52.000,A 180.000,B 0.000,C 180.000} C_DIS
LIN {X 106.669,Y 8.405,Z 52.000,A 180.000,B 0.000,C 180.000} C_DIS
LIN {X 106.550,Y 8.355,Z 52.000,A 180.000,B 0.000,C 180.000} C_DIS
LIN {X 105.120,Y 7.773,Z 52.000,A 180.000,B 0.000,C 180.000} C_DIS
LIN {X 104.941,Y 7.701,Z 52.000,A 180.000,B 0.000,C 180.000} C_DIS
LIN {X 103.504,Y 7.154,Z 52.000,A 180.000,B 0.000,C 180.000} C_DIS
LIN {X 103.332,Y 7.089,Z 52.000,A 180.000,B 0.000,C 180.000} C_DIS
LIN {X 103.153,Y 7.026,Z 52.000,A 180.000,B 0.000,C 180.000} C_DIS
LIN {X 101.723,Y 6.520,Z 52.000,A 180.000,B 0.000,C 180.000} C_DIS
LIN {X 101.545,Y 6.460,Z 52.000,A 180.000,B 0.000,C 180.000} C_DIS
LIN {X 100.114,Y 5.992,Z 52.000,A 180.000,B 0.000,C 180.000} C_DIS
LIN {X 99.936,Y 5.935,Z 52.000,A 180.000,B 0.000,C 180.000} C_DIS
LIN {X 98.505,Y 5.503,Z 52.000,A 180.000,B 0.000,C 180.000} C_DIS
LIN {X 98.327,Y 5.450,Z 52.000,A 180.000,B 0.000,C 180.000} C_DIS
LIN {X 98.148,Y 5.400,Z 52.000,A 180.000,B 0.000,C 180.000} C_DIS
LIN {X 96.718,Y 5.005,Z 52.000,A 180.000,B 0.000,C 180.000} C_DIS
LIN {X 96.539,Y 4.958,Z 52.000,A 180.000,B 0.000,C 180.000} C_DIS
LIN {X 95.109,Y 4.598,Z 52.000,A 180.000,B 0.000,C 180.000} C_DIS
LIN {X 94.930,Y 4.554,Z 52.000,A 180.000,B 0.000,C 180.000} C_DIS
LIN {X 94.751,Y 4.513,Z 52.000,A 180.000,B 0.000,C 180.000} C_DIS
LIN {X 93.321,Y 4.189,Z 52.000,A 180.000,B 0.000,C 180.000} C_DIS
LIN {X 93.142,Y 4.150,Z 52.000,A 180.000,B 0.000,C 180.000} C_DIS
LIN {X 91.533,Y 3.825,Z 52.000,A 180.000,B 0.000,C 180.000} C_DIS
LIN {X 91.355,Y 3.792,Z 52.000,A 180.000,B 0.000,C 180.000} C_DIS
LIN {X 89.925,Y 3.538,Z 52.000,A 180.000,B 0.000,C 180.000} C_DIS
LIN {X 89.746,Y 3.506,Z 52.000,A 180.000,B 0.000,C 180.000} C_DIS
LIN {X 89.567,Y 3.479,Z 52.000,A 180.000,B 0.000,C 180.000} C_DIS
LIN {X 88.137,Y 3.259,Z 52.000,A 180.000,B 0.000,C 180.000} C_DIS
LIN {X 87.958,Y 3.233,Z 52.000,A 180.000,B 0.000,C 180.000} C_DIS
LIN {X 86.349,Y 3.025,Z 52.000,A 180.000,B 0.000,C 180.000} C_DIS
LIN {X 86.170,Y 3.004,Z 52.000,A 180.000,B 0.000,C 180.000} C_DIS
LIN {X 84.561,Y 2.833,Z 52.000,A 180.000,B 0.000,C 180.000} C_DIS
LIN {X 84.383,Y 2.818,Z 52.000,A 180.000,B 0.000,C 180.000} C_DIS
LIN {X 82.952,Y 2.700,Z 52.000,A 180.000,B 0.000,C 180.000} C_DIS
LIN {X 82.774,Y 2.686,Z 52.000,A 180.000,B 0.000,C 180.000} C_DIS
LIN {X 82.761,Y 2.685,Z 52.000,A 180.000,B 0.000,C 180.000} C_DIS
LIN {X 82.595,Y 2.675,Z 52.000,A 180.000,B 0.000,C 180.000} C_DIS
LIN {X 81.165,Y 2.591,Z 52.000,A 180.000,B 0.000,C 180.000} C_DIS
LIN {X 80.986,Y 2.581,Z 52.000,A 180.000,B 0.000,C 180.000} C_DIS
LIN {X 79.377,Y 2.525,Z 52.000,A 180.000,B 0.000,C 180.000} C_DIS
LIN {X 79.198,Y 2.520,Z 52.000,A 180.000,B 0.000,C 180.000} C_DIS
LIN {X 77.589,Y 2.501,Z 52.000,A 180.000,B 0.000,C 180.000} C_DIS
LIN {X 77.411,Y 2.501,Z 52.000,A 180.000,B 0.000,C 180.000} C_DIS
LIN {X 75.802,Y 2.520,Z 52.000,A 180.000,B 0.000,C 180.000} C_DIS
LIN {X 75.623,Y 2.525,Z 52.000,A 180.000,B 0.000,C 180.000} C_DIS
LIN {X 74.014,Y 2.581,Z 52.000,A 180.000,B 0.000,C 180.000} C_DIS
LIN {X 73.835,Y 2.591,Z 52.000,A 180.000,B 0.000,C 180.000} C_DIS
LIN {X 72.405,Y 2.675,Z 52.000,A 180.000,B 0.000,C 180.000} C_DIS
LIN {X 72.239,Y 2.685,Z 52.000,A 180.000,B 0.000,C 180.000} C_DIS
LIN {X 72.226,Y 2.686,Z 52.000,A 180.000,B 0.000,C 180.000} C_DIS
LIN {X 72.048,Y 2.700,Z 52.000,A 180.000,B 0.000,C 180.000} C_DIS
LIN {X 70.617,Y 2.818,Z 52.000,A 180.000,B 0.000,C 180.000} C_DIS
LIN {X 70.439,Y 2.833,Z 52.000,A 180.000,B 0.000,C 180.000} C_DIS
LIN {X 68.830,Y 3.004,Z 52.000,A 180.000,B 0.000,C 180.000} C_DIS
LIN {X 68.651,Y 3.025,Z 52.000,A 180.000,B 0.000,C 180.000} C_DIS
LIN {X 67.042,Y 3.233,Z 52.000,A 180.000,B 0.000,C 180.000} C_DIS
LIN {X 66.863,Y 3.259,Z 52.000,A 180.000,B 0.000,C 180.000} C_DIS
LIN {X 65.433,Y 3.479,Z 52.000,A 180.000,B 0.000,C 180.000} C_DIS
LIN {X 65.254,Y 3.506,Z 52.000,A 180.000,B 0.000,C 180.000} C_DIS
LIN {X 65.075,Y 3.538,Z 52.000,A 180.000,B 0.000,C 180.000} C_DIS
LIN {X 63.645,Y 3.792,Z 52.000,A 180.000,B 0.000,C 180.000} C_DIS
LIN {X 63.467,Y 3.825,Z 52.000,A 180.000,B 0.000,C 180.000} C_DIS
LIN {X 61.858,Y 4.150,Z 52.000,A 180.000,B 0.000,C 180.000} C_DIS
LIN {X 61.679,Y 4.189,Z 52.000,A 180.000,B 0.000,C 180.000} C_DIS
LIN {X 60.249,Y 4.513,Z 52.000,A 180.000,B 0.000,C 180.000} C_DIS
LIN {X 60.070,Y 4.554,Z 52.000,A 180.000,B 0.000,C 180.000} C_DIS
LIN {X 59.891,Y 4.598,Z 52.000,A 180.000,B 0.000,C 180.000} C_DIS
LIN {X 58.461,Y 4.958,Z 52.000,A 180.000,B 0.000,C 180.000} C_DIS
LIN {X 58.282,Y 5.005,Z 52.000,A 180.000,B 0.000,C 180.000} C_DIS
LIN {X 56.852,Y 5.400,Z 52.000,A 180.000,B 0.000,C 180.000} C_DIS
LIN {X 56.673,Y 5.450,Z 52.000,A 180.000,B 0.000,C 180.000} C_DIS
LIN {X 56.495,Y 5.503,Z 52.000,A 180.000,B 0.000,C 180.000} C_DIS
LIN {X 55.064,Y 5.935,Z 52.000,A 180.000,B 0.000,C 180.000} C_DIS
LIN {X 54.886,Y 5.992,Z 52.000,A 180.000,B 0.000,C 180.000} C_DIS
LIN {X 53.455,Y 6.460,Z 52.000,A 180.000,B 0.000,C 180.000} C_DIS
LIN {X 53.277,Y 6.520,Z 52.000,A 180.000,B 0.000,C 180.000} C_DIS
LIN {X 51.847,Y 7.026,Z 52.000,A 180.000,B 0.000,C 180.000} C_DIS
LIN {X 51.668,Y 7.089,Z 52.000,A 180.000,B 0.000,C 180.000} C_DIS
LIN {X 51.496,Y 7.154,Z 52.000,A 180.000,B 0.000,C 180.000} C_DIS
LIN {X 50.059,Y 7.701,Z 52.000,A 180.000,B 0.000,C 180.000} C_DIS
LIN {X 49.880,Y 7.773,Z 52.000,A 180.000,B 0.000,C 180.000} C_DIS
LIN {X 48.450,Y 8.355,Z 52.000,A 180.000,B 0.000,C 180.000} C_DIS
LIN {X 48.331,Y 8.405,Z 52.000,A 180.000,B 0.000,C 180.000} C_DIS
LIN {X 46.841,Y 9.053,Z 52.000,A 180.000,B 0.000,C 180.000} C_DIS
LIN {X 46.692,Y 9.120,Z 52.000,A 180.000,B 0.000,C 180.000} C_DIS
LIN {X 45.232,Y 9.797,Z 52.000,A 180.000,B 0.000,C 180.000} C_DIS
LIN {X 45.151,Y 9.836,Z 52.000,A 180.000,B 0.000,C 180.000} C_DIS
LIN {X 43.697,Y 10.551,Z 52.000,A 180.000,B 0.000,C 180.000} C_DIS
LIN {X 43.623,Y 10.587,Z 52.000,A 180.000,B 0.000,C 180.000} C_DIS
LIN {X 43.444,Y 10.680,Z 52.000,A 180.000,B 0.000,C 180.000} C_DIS
LIN {X 42.193,Y 11.332,Z 52.000,A 180.000,B 0.000,C 180.000} C_DIS
LIN {X 42.014,Y 11.426,Z 52.000,A 180.000,B 0.000,C 180.000} C_DIS
LIN {X 40.584,Y 12.215,Z 52.000,A 180.000,B 0.000,C 180.000} C_DIS
LIN {X 40.405,Y 12.317,Z 52.000,A 180.000,B 0.000,C 180.000} C_DIS
LIN {X 39.141,Y 13.053,Z 52.000,A 180.000,B 0.000,C 180.000} C_DIS
LIN {X 38.975,Y 13.151,Z 52.000,A 180.000,B 0.000,C 180.000} C_DIS
LIN {X 38.842,Y 13.232,Z 52.000,A 180.000,B 0.000,C 180.000} C_DIS
LIN {X 37.545,Y 14.029,Z 52.000,A 180.000,B 0.000,C 180.000} C_DIS
LIN {X 37.393,Y 14.126,Z 52.000,A 180.000,B 0.000,C 180.000} C_DIS
LIN {X 36.115,Y 14.953,Z 52.000,A 180.000,B 0.000,C 180.000} C_DIS
LIN {X 36.012,Y 15.020,Z 52.000,A 180.000,B 0.000,C 180.000} C_DIS
LIN {X 35.936,Y 15.072,Z 52.000,A 180.000,B 0.000,C 180.000} C_DIS
LIN {X 34.685,Y 15.924,Z 52.000,A 180.000,B 0.000,C 180.000} C_DIS
LIN {X 34.506,Y 16.047,Z 52.000,A 180.000,B 0.000,C 180.000} C_DIS
LIN {X 33.194,Y 16.986,Z 52.000,A 180.000,B 0.000,C 180.000} C_DIS
LIN {X 33.076,Y 17.073,Z 52.000,A 180.000,B 0.000,C 180.000} C_DIS
LIN {X 31.765,Y 18.059,Z 52.000,A 180.000,B 0.000,C 180.000} C_DIS
LIN {X 31.646,Y 18.152,Z 52.000,A 180.000,B 0.000,C 180.000} C_DIS
LIN {X 30.394,Y 19.139,Z 52.000,A 180.000,B 0.000,C 180.000} C_DIS
LIN {X 30.215,Y 19.286,Z 52.000,A 180.000,B 0.000,C 180.000} C_DIS
LIN {X 29.106,Y 20.204,Z 52.000,A 180.000,B 0.000,C 180.000} C_DIS
LIN {X 28.964,Y 20.323,Z 52.000,A 180.000,B 0.000,C 180.000} C_DIS
LIN {X 27.713,Y 21.410,Z 52.000,A 180.000,B 0.000,C 180.000} C_DIS
LIN {X 27.660,Y 21.456,Z 52.000,A 180.000,B 0.000,C 180.000} C_DIS
LIN {X 27.534,Y 21.570,Z 52.000,A 180.000,B 0.000,C 180.000} C_DIS
LIN {X 26.461,Y 22.547,Z 52.000,A 180.000,B 0.000,C 180.000} C_DIS
LIN {X 26.289,Y 22.707,Z 52.000,A 180.000,B 0.000,C 180.000} C_DIS
LIN {X 25.165,Y 23.780,Z 52.000,A 180.000,B 0.000,C 180.000} C_DIS
LIN {X 25.031,Y 23.910,Z 52.000,A 180.000,B 0.000,C 180.000} C_DIS
LIN {X 23.910,Y 25.031,Z 52.000,A 180.000,B 0.000,C 180.000} C_DIS
LIN {X 23.780,Y 25.165,Z 52.000,A 180.000,B 0.000,C 180.000} C_DIS
LIN {X 22.707,Y 26.289,Z 52.000,A 180.000,B 0.000,C 180.000} C_DIS
LIN {X 22.547,Y 26.461,Z 52.000,A 180.000,B 0.000,C 180.000} C_DIS
LIN {X 21.570,Y 27.534,Z 52.000,A 180.000,B 0.000,C 180.000} C_DIS
LIN {X 21.456,Y 27.660,Z 52.000,A 180.000,B 0.000,C 180.000} C_DIS
LIN {X 21.410,Y 27.713,Z 52.000,A 180.000,B 0.000,C 180.000} C_DIS
LIN {X 20.323,Y 28.964,Z 52.000,A 180.000,B 0.000,C 180.000} C_DIS
LIN {X 20.204,Y 29.106,Z 52.000,A 180.000,B 0.000,C 180.000} C_DIS
LIN {X 19.286,Y 30.215,Z 52.000,A 180.000,B 0.000,C 180.000} C_DIS
LIN {X 19.139,Y 30.394,Z 52.000,A 180.000,B 0.000,C 180.000} C_DIS
LIN {X 18.152,Y 31.646,Z 52.000,A 180.000,B 0.000,C 180.000} C_DIS
LIN {X 18.059,Y 31.765,Z 52.000,A 180.000,B 0.000,C 180.000} C_DIS
LIN {X 17.073,Y 33.076,Z 52.000,A 180.000,B 0.000,C 180.000} C_DIS
LIN {X 16.986,Y 33.194,Z 52.000,A 180.000,B 0.000,C 180.000} C_DIS
LIN {X 16.047,Y 34.506,Z 52.000,A 180.000,B 0.000,C 180.000} C_DIS
LIN {X 15.924,Y 34.685,Z 52.000,A 180.000,B 0.000,C 180.000} C_DIS
LIN {X 15.072,Y 35.936,Z 52.000,A 180.000,B 0.000,C 180.000} C_DIS
LIN {X 15.020,Y 36.012,Z 52.000,A 180.000,B 0.000,C 180.000} C_DIS
LIN {X 14.953,Y 36.115,Z 52.000,A 180.000,B 0.000,C 180.000} C_DIS
LIN {X 14.126,Y 37.393,Z 52.000,A 180.000,B 0.000,C 180.000} C_DIS
LIN {X 14.029,Y 37.545,Z 52.000,A 180.000,B 0.000,C 180.000} C_DIS
LIN {X 13.232,Y 38.842,Z 52.000,A 180.000,B 0.000,C 180.000} C_DIS
LIN {X 13.151,Y 38.975,Z 52.000,A 180.000,B 0.000,C 180.000} C_DIS
LIN {X 13.053,Y 39.141,Z 52.000,A 180.000,B 0.000,C 180.000} C_DIS
LIN {X 12.317,Y 40.405,Z 52.000,A 180.000,B 0.000,C 180.000} C_DIS
LIN {X 12.215,Y 40.584,Z 52.000,A 180.000,B 0.000,C 180.000} C_DIS
LIN {X 11.426,Y 42.014,Z 52.000,A 180.000,B 0.000,C 180.000} C_DIS
LIN {X 11.332,Y 42.193,Z 52.000,A 180.000,B 0.000,C 180.000} C_DIS
LIN {X 10.680,Y 43.444,Z 52.000,A 180.000,B 0.000,C 180.000} C_DIS
LIN {X 10.587,Y 43.623,Z 52.000,A 180.000,B 0.000,C 180.000} C_DIS
LIN {X 10.551,Y 43.697,Z 52.000,A 180.000,B 0.000,C 180.000} C_DIS
LIN {X 9.836,Y 45.151,Z 52.000,A 180.000,B 0.000,C 180.000} C_DIS
LIN {X 9.797,Y 45.232,Z 52.000,A 180.000,B 0.000,C 180.000} C_DIS
LIN {X 9.120,Y 46.692,Z 52.000,A 180.000,B 0.000,C 180.000} C_DIS
LIN {X 9.053,Y 46.841,Z 52.000,A 180.000,B 0.000,C 180.000} C_DIS
LIN {X 8.405,Y 48.331,Z 52.000,A 180.000,B 0.000,C 180.000} C_DIS
LIN {X 8.355,Y 48.450,Z 52.000,A 180.000,B 0.000,C 180.000} C_DIS
LIN {X 7.773,Y 49.880,Z 52.000,A 180.000,B 0.000,C 180.000} C_DIS
LIN {X 7.701,Y 50.059,Z 52.000,A 180.000,B 0.000,C 180.000} C_DIS
LIN {X 7.154,Y 51.496,Z 52.000,A 180.000,B 0.000,C 180.000} C_DIS
LIN {X 7.089,Y 51.668,Z 52.000,A 180.000,B 0.000,C 180.000} C_DIS
